    CONST robtarget p12664:= [[1532.1310620615823, -51.755404230859114, 1003.500033578516], [0, 0, 1, 0], [0, 0, 0, 0], [9E9, 9E9, 9E9, 9E9, 9E9, 9E9]];
    CONST robtarget p12665:= [[1531.2618371973992, -52.270415118434464, 1003.500033578516], [0, 0, 1, 0], [0, 0, 0, 0], [9E9, 9E9, 9E9, 9E9, 9E9, 9E9]];
    CONST robtarget p12666:= [[1530.6100576659546, -52.63207456238566, 1003.500033578516], [0, 0, 1, 0], [0, 0, 0, 0], [9E9, 9E9, 9E9, 9E9, 9E9, 9E9]];
    CONST robtarget p12667:= [[1530.2931638971058, -52.82618686460231, 1003.500033578516], [0, 0, 1, 0], [0, 0, 0, 0], [9E9, 9E9, 9E9, 9E9, 9E9, 9E9]];
    CONST robtarget p12668:= [[1529.7863810110655, -53.08892651938235, 1003.500033578516], [0, 0, 1, 0], [0, 0, 0, 0], [9E9, 9E9, 9E9, 9E9, 9E9, 9E9]];
    CONST robtarget p12669:= [[1529.7367415978995, -53.11810760441107, 1003.500033578516], [0, 0, 1, 0], [0, 0, 0, 0], [9E9, 9E9, 9E9, 9E9, 9E9, 9E9]];
    CONST robtarget p12670:= [[1529.1847719882317, -53.41718675288824, 1003.500033578516], [0, 0, 1, 0], [0, 0, 0, 0], [9E9, 9E9, 9E9, 9E9, 9E9, 9E9]];
    CONST robtarget p12671:= [[1528.9656328563278, -53.54211952816121, 1003.500033578516], [0, 0, 1, 0], [0, 0, 0, 0], [9E9, 9E9, 9E9, 9E9, 9E9, 9E9]];
    CONST robtarget p12672:= [[1528.4780900744865, -53.83944066606885, 1003.500033578516], [0, 0, 1, 0], [0, 0, 0, 0], [9E9, 9E9, 9E9, 9E9, 9E9, 9E9]];
    CONST robtarget p12673:= [[1527.6960366206135, -54.26689992615866, 1003.500033578516], [0, 0, 1, 0], [0, 0, 0, 0], [9E9, 9E9, 9E9, 9E9, 9E9, 9E9]];
    CONST robtarget p12674:= [[1527.2898060617083, -54.45592588754269, 1003.500033578516], [0, 0, 1, 0], [0, 0, 0, 0], [9E9, 9E9, 9E9, 9E9, 9E9, 9E9]];
    CONST robtarget p12675:= [[1526.7303787533363, -54.710685409871346, 1003.500033578516], [0, 0, 1, 0], [0, 0, 0, 0], [9E9, 9E9, 9E9, 9E9, 9E9, 9E9]];
    CONST robtarget p12676:= [[1526.1686464097916, -54.92872139464171, 1003.500033578516], [0, 0, 1, 0], [0, 0, 0, 0], [9E9, 9E9, 9E9, 9E9, 9E9, 9E9]];
    CONST robtarget p12677:= [[1525.7512622465076, -55.13249219015158, 1003.500033578516], [0, 0, 1, 0], [0, 0, 0, 0], [9E9, 9E9, 9E9, 9E9, 9E9, 9E9]];
    CONST robtarget p12678:= [[1525.1590179163616, -55.431827644455886, 1003.500033578516], [0, 0, 1, 0], [0, 0, 0, 0], [9E9, 9E9, 9E9, 9E9, 9E9, 9E9]];
    CONST robtarget p12679:= [[1525.0064466097315, -55.5144084202345, 1003.500033578516], [0, 0, 1, 0], [0, 0, 0, 0], [9E9, 9E9, 9E9, 9E9, 9E9, 9E9]];
    CONST robtarget p12680:= [[1524.838681406511, -55.59887141094046, 1003.500033578516], [0, 0, 1, 0], [0, 0, 0, 0], [9E9, 9E9, 9E9, 9E9, 9E9, 9E9]];
    CONST robtarget p12681:= [[1524.412701120568, -55.80300474395773, 1003.500033578516], [0, 0, 1, 0], [0, 0, 0, 0], [9E9, 9E9, 9E9, 9E9, 9E9, 9E9]];
    CONST robtarget p12682:= [[1523.8137863507948, -56.0413945246957, 1003.500033578516], [0, 0, 1, 0], [0, 0, 0, 0], [9E9, 9E9, 9E9, 9E9, 9E9, 9E9]];
    CONST robtarget p12683:= [[1523.096794661028, -56.341017791955295, 1003.500033578516], [0, 0, 1, 0], [0, 0, 0, 0], [9E9, 9E9, 9E9, 9E9, 9E9, 9E9]];
    CONST robtarget p12684:= [[1522.900783238865, -56.42082180491421, 1003.500033578516], [0, 0, 1, 0], [0, 0, 0, 0], [9E9, 9E9, 9E9, 9E9, 9E9, 9E9]];
    CONST robtarget p12685:= [[1522.6082814196384, -56.545971688333516, 1003.500033578516], [0, 0, 1, 0], [0, 0, 0, 0], [9E9, 9E9, 9E9, 9E9, 9E9, 9E9]];
    CONST robtarget p12686:= [[1522.1889282350046, -56.6709628567649, 1003.500033578516], [0, 0, 1, 0], [0, 0, 0, 0], [9E9, 9E9, 9E9, 9E9, 9E9, 9E9]];
    CONST robtarget p12687:= [[1521.3015503338331, -57.03764612699189, 1003.500033578516], [0, 0, 1, 0], [0, 0, 0, 0], [9E9, 9E9, 9E9, 9E9, 9E9, 9E9]];
    CONST robtarget p12688:= [[1520.80306051841, -57.23276139857534, 1003.500033578516], [0, 0, 1, 0], [0, 0, 0, 0], [9E9, 9E9, 9E9, 9E9, 9E9, 9E9]];
    CONST robtarget p12689:= [[1520.6617507120266, -57.27868779379712, 1003.500033578516], [0, 0, 1, 0], [0, 0, 0, 0], [9E9, 9E9, 9E9, 9E9, 9E9, 9E9]];
    CONST robtarget p12690:= [[1519.8184170172012, -57.589773311048475, 1003.500033578516], [0, 0, 1, 0], [0, 0, 0, 0], [9E9, 9E9, 9E9, 9E9, 9E9, 9E9]];
    CONST robtarget p12691:= [[1519.6469440456822, -57.65315375966382, 1003.500033578516], [0, 0, 1, 0], [0, 0, 0, 0], [9E9, 9E9, 9E9, 9E9, 9E9, 9E9]];
    CONST robtarget p12692:= [[1518.9672123317812, -57.88370126778568, 1003.500033578516], [0, 0, 1, 0], [0, 0, 0, 0], [9E9, 9E9, 9E9, 9E9, 9E9, 9E9]];
    CONST robtarget p12693:= [[1517.866507887685, -58.20960162710837, 1003.500033578516], [0, 0, 1, 0], [0, 0, 0, 0], [9E9, 9E9, 9E9, 9E9, 9E9, 9E9]];
    CONST robtarget p12694:= [[1517.564370643482, -58.28325027030423, 1003.500033578516], [0, 0, 1, 0], [0, 0, 0, 0], [9E9, 9E9, 9E9, 9E9, 9E9, 9E9]];
    CONST robtarget p12695:= [[1517.3151101543563, -58.359110977004875, 1003.500033578516], [0, 0, 1, 0], [0, 0, 0, 0], [9E9, 9E9, 9E9, 9E9, 9E9, 9E9]];
    CONST robtarget p12696:= [[1516.4046109578076, -58.64286422475155, 1003.500033578516], [0, 0, 1, 0], [0, 0, 0, 0], [9E9, 9E9, 9E9, 9E9, 9E9, 9E9]];
    CONST robtarget p12697:= [[1515.9569505437983, -58.768392762982955, 1003.500033578516], [0, 0, 1, 0], [0, 0, 0, 0], [9E9, 9E9, 9E9, 9E9, 9E9, 9E9]];
    CONST robtarget p12698:= [[1515.5151199352963, -58.91022808552202, 1003.500033578516], [0, 0, 1, 0], [0, 0, 0, 0], [9E9, 9E9, 9E9, 9E9, 9E9, 9E9]];
    CONST robtarget p12699:= [[1515.192527778176, -58.960963909001194, 1003.500033578516], [0, 0, 1, 0], [0, 0, 0, 0], [9E9, 9E9, 9E9, 9E9, 9E9, 9E9]];
    CONST robtarget p12700:= [[1514.1503402686096, -59.22694543179028, 1003.500033578516], [0, 0, 1, 0], [0, 0, 0, 0], [9E9, 9E9, 9E9, 9E9, 9E9, 9E9]];
    CONST robtarget p12701:= [[1513.5557447633169, -59.360352740508816, 1003.500033578516], [0, 0, 1, 0], [0, 0, 0, 0], [9E9, 9E9, 9E9, 9E9, 9E9, 9E9]];
    CONST robtarget p12702:= [[1513.2934993638064, -59.398941220659864, 1003.500033578516], [0, 0, 1, 0], [0, 0, 0, 0], [9E9, 9E9, 9E9, 9E9, 9E9, 9E9]];
    CONST robtarget p12703:= [[1512.403489281292, -59.608763300548, 1003.500033578516], [0, 0, 1, 0], [0, 0, 0, 0], [9E9, 9E9, 9E9, 9E9, 9E9, 9E9]];
    CONST robtarget p12704:= [[1512.0296429570128, -59.685111800334646, 1003.500033578516], [0, 0, 1, 0], [0, 0, 0, 0], [9E9, 9E9, 9E9, 9E9, 9E9, 9E9]];
    CONST robtarget p12705:= [[1511.4338776805575, -59.82476628793355, 1003.500033578516], [0, 0, 1, 0], [0, 0, 0, 0], [9E9, 9E9, 9E9, 9E9, 9E9, 9E9]];
    CONST robtarget p12706:= [[1510.9881098887731, -59.91814747321601, 1003.500033578516], [0, 0, 1, 0], [0, 0, 0, 0], [9E9, 9E9, 9E9, 9E9, 9E9, 9E9]];
    CONST robtarget p12707:= [[1510.8070079036906, -59.94973532784152, 1003.500033578516], [0, 0, 1, 0], [0, 0, 0, 0], [9E9, 9E9, 9E9, 9E9, 9E9, 9E9]];
    CONST robtarget p12708:= [[1510.7448277760268, -59.96038495608518, 1003.500033578516], [0, 0, 1, 0], [0, 0, 0, 0], [9E9, 9E9, 9E9, 9E9, 9E9, 9E9]];
    CONST robtarget p12709:= [[1510.4745015685621, -59.98646378804859, 1003.500033578516], [0, 0, 1, 0], [0, 0, 0, 0], [9E9, 9E9, 9E9, 9E9, 9E9, 9E9]];
    CONST robtarget p12710:= [[1510.0909268709627, -60.04140453241323, 1003.500033578516], [0, 0, 1, 0], [0, 0, 0, 0], [9E9, 9E9, 9E9, 9E9, 9E9, 9E9]];
    CONST robtarget p12711:= [[1509.4092115213996, -60.151023493626894, 1003.500033578516], [0, 0, 1, 0], [0, 0, 0, 0], [9E9, 9E9, 9E9, 9E9, 9E9, 9E9]];
    CONST robtarget p12712:= [[1509.1407802614508, -60.19882687326773, 1003.500033578516], [0, 0, 1, 0], [0, 0, 0, 0], [9E9, 9E9, 9E9, 9E9, 9E9, 9E9]];
    CONST robtarget p12713:= [[1508.5601837016875, -60.26340042336168, 1003.500033578516], [0, 0, 1, 0], [0, 0, 0, 0], [9E9, 9E9, 9E9, 9E9, 9E9, 9E9]];
    CONST robtarget p12714:= [[1507.6640295886964, -60.397835897292495, 1003.500033578516], [0, 0, 1, 0], [0, 0, 0, 0], [9E9, 9E9, 9E9, 9E9, 9E9, 9E9]];
    CONST robtarget p12715:= [[1507.3205366995528, -60.44744484086121, 1003.500033578516], [0, 0, 1, 0], [0, 0, 0, 0], [9E9, 9E9, 9E9, 9E9, 9E9, 9E9]];
    CONST robtarget p12716:= [[1506.9198397004645, -60.48554848075174, 1003.500033578516], [0, 0, 1, 0], [0, 0, 0, 0], [9E9, 9E9, 9E9, 9E9, 9E9, 9E9]];
    CONST robtarget p12717:= [[1506.3480021439116, -60.54932865497324, 1003.500033578516], [0, 0, 1, 0], [0, 0, 0, 0], [9E9, 9E9, 9E9, 9E9, 9E9, 9E9]];
    CONST robtarget p12718:= [[1506.0286245296538, -60.606260280640186, 1003.500033578516], [0, 0, 1, 0], [0, 0, 0, 0], [9E9, 9E9, 9E9, 9E9, 9E9, 9E9]];
    CONST robtarget p12719:= [[1505.9492369877419, -60.60951490106271, 1003.500033578516], [0, 0, 1, 0], [0, 0, 0, 0], [9E9, 9E9, 9E9, 9E9, 9E9, 9E9]];
    CONST robtarget p12720:= [[1505.8789526524727, -60.611009085656356, 1003.500033578516], [0, 0, 1, 0], [0, 0, 0, 0], [9E9, 9E9, 9E9, 9E9, 9E9, 9E9]];
    CONST robtarget p12721:= [[1505.3224203883021, -60.65045746650896, 1003.500033578516], [0, 0, 1, 0], [0, 0, 0, 0], [9E9, 9E9, 9E9, 9E9, 9E9, 9E9]];
    CONST robtarget p12722:= [[1505.1441541680317, -60.672558378263645, 1003.500033578516], [0, 0, 1, 0], [0, 0, 0, 0], [9E9, 9E9, 9E9, 9E9, 9E9, 9E9]];
    CONST robtarget p12723:= [[1504.3770680072512, -60.70421225380319, 1003.500033578516], [0, 0, 1, 0], [0, 0, 0, 0], [9E9, 9E9, 9E9, 9E9, 9E9, 9E9]];
    CONST robtarget p12724:= [[1503.8992364217452, -60.77229114782248, 1003.500033578516], [0, 0, 1, 0], [0, 0, 0, 0], [9E9, 9E9, 9E9, 9E9, 9E9, 9E9]];
    CONST robtarget p12725:= [[1503.093503312446, -60.829713664428, 1003.500033578516], [0, 0, 1, 0], [0, 0, 0, 0], [9E9, 9E9, 9E9, 9E9, 9E9, 9E9]];
    CONST robtarget p12726:= [[1502.275028322799, -60.865266701102776, 1003.500033578516], [0, 0, 1, 0], [0, 0, 0, 0], [9E9, 9E9, 9E9, 9E9, 9E9, 9E9]];
    CONST robtarget p12727:= [[1501.7502801780977, -60.87680720154429, 1003.500033578516], [0, 0, 1, 0], [0, 0, 0, 0], [9E9, 9E9, 9E9, 9E9, 9E9, 9E9]];
    CONST robtarget p12728:= [[1501.1321717850142, -60.86812155272374, 1003.500033578516], [0, 0, 1, 0], [0, 0, 0, 0], [9E9, 9E9, 9E9, 9E9, 9E9, 9E9]];
    CONST robtarget p12729:= [[1500.3650176022602, -60.89439954561838, 1003.500033578516], [0, 0, 1, 0], [0, 0, 0, 0], [9E9, 9E9, 9E9, 9E9, 9E9, 9E9]];
    CONST robtarget p12730:= [[1500.0005887741925, -60.88714554662218, 1003.500033578516], [0, 0, 1, 0], [0, 0, 0, 0], [9E9, 9E9, 9E9, 9E9, 9E9, 9E9]];
    CONST robtarget p12731:= [[1499.6330786731016, -60.86918679644523, 1003.500033578516], [0, 0, 1, 0], [0, 0, 0, 0], [9E9, 9E9, 9E9, 9E9, 9E9, 9E9]];
    CONST robtarget p12732:= [[1498.7343183829123, -60.89301213573544, 1003.500033578516], [0, 0, 1, 0], [0, 0, 0, 0], [9E9, 9E9, 9E9, 9E9, 9E9, 9E9]];
    CONST robtarget p12733:= [[1497.8384561952996, -60.879011023600654, 1003.500033578516], [0, 0, 1, 0], [0, 0, 0, 0], [9E9, 9E9, 9E9, 9E9, 9E9, 9E9]];
    CONST robtarget p12734:= [[1497.0922041448482, -60.83771003512446, 1003.500033578516], [0, 0, 1, 0], [0, 0, 0, 0], [9E9, 9E9, 9E9, 9E9, 9E9, 9E9]];
    CONST robtarget p12735:= [[1496.8361997453076, -60.82603686445868, 1003.500033578516], [0, 0, 1, 0], [0, 0, 0, 0], [9E9, 9E9, 9E9, 9E9, 9E9, 9E9]];
    CONST robtarget p12736:= [[1496.4138965917214, -60.778275502153924, 1003.500033578516], [0, 0, 1, 0], [0, 0, 0, 0], [9E9, 9E9, 9E9, 9E9, 9E9, 9E9]];
    CONST robtarget p12737:= [[1495.8035146590512, -60.74767869639028, 1003.500033578516], [0, 0, 1, 0], [0, 0, 0, 0], [9E9, 9E9, 9E9, 9E9, 9E9, 9E9]];
    CONST robtarget p12738:= [[1495.6187393990072, -60.72769177277266, 1003.500033578516], [0, 0, 1, 0], [0, 0, 0, 0], [9E9, 9E9, 9E9, 9E9, 9E9, 9E9]];
    CONST robtarget p12739:= [[1495.126932201303, -60.70252857016523, 1003.500033578516], [0, 0, 1, 0], [0, 0, 0, 0], [9E9, 9E9, 9E9, 9E9, 9E9, 9E9]];
    CONST robtarget p12740:= [[1494.505248273516, -60.640040835068014, 1003.500033578516], [0, 0, 1, 0], [0, 0, 0, 0], [9E9, 9E9, 9E9, 9E9, 9E9, 9E9]];
    CONST robtarget p12741:= [[1493.9707970922311, -60.586603258026315, 1003.500033578516], [0, 0, 1, 0], [0, 0, 0, 0], [9E9, 9E9, 9E9, 9E9, 9E9, 9E9]];
    CONST robtarget p12742:= [[1493.728122281413, -60.57869577579727, 1003.500033578516], [0, 0, 1, 0], [0, 0, 0, 0], [9E9, 9E9, 9E9, 9E9, 9E9, 9E9]];
    CONST robtarget p12743:= [[1493.3207496594594, -60.545796007754376, 1003.500033578516], [0, 0, 1, 0], [0, 0, 0, 0], [9E9, 9E9, 9E9, 9E9, 9E9, 9E9]];
    CONST robtarget p12744:= [[1493.0342588648045, -60.515907015423046, 1003.500033578516], [0, 0, 1, 0], [0, 0, 0, 0], [9E9, 9E9, 9E9, 9E9, 9E9, 9E9]];
    CONST robtarget p12745:= [[1492.5314490561839, -60.42360355630814, 1003.500033578516], [0, 0, 1, 0], [0, 0, 0, 0], [9E9, 9E9, 9E9, 9E9, 9E9, 9E9]];
    CONST robtarget p12746:= [[1491.6668361516013, -60.32164521258506, 1003.500033578516], [0, 0, 1, 0], [0, 0, 0, 0], [9E9, 9E9, 9E9, 9E9, 9E9, 9E9]];
    CONST robtarget p12747:= [[1490.7479630489497, -60.18407184896695, 1003.500033578516], [0, 0, 1, 0], [0, 0, 0, 0], [9E9, 9E9, 9E9, 9E9, 9E9, 9E9]];
    CONST robtarget p12748:= [[1489.9914983282804, -60.0648048675663, 1003.500033578516], [0, 0, 1, 0], [0, 0, 0, 0], [9E9, 9E9, 9E9, 9E9, 9E9, 9E9]];
    CONST robtarget p12749:= [[1489.8132747932655, -60.050032149975266, 1003.500033578516], [0, 0, 1, 0], [0, 0, 0, 0], [9E9, 9E9, 9E9, 9E9, 9E9, 9E9]];
    CONST robtarget p12750:= [[1489.6954944579838, -60.02336426978388, 1003.500033578516], [0, 0, 1, 0], [0, 0, 0, 0], [9E9, 9E9, 9E9, 9E9, 9E9, 9E9]];
    CONST robtarget p12751:= [[1489.2307032090532, -59.94463917957851, 1003.500033578516], [0, 0, 1, 0], [0, 0, 0, 0], [9E9, 9E9, 9E9, 9E9, 9E9, 9E9]];
    CONST robtarget p12752:= [[1488.969375621922, -59.912737352572954, 1003.500033578516], [0, 0, 1, 0], [0, 0, 0, 0], [9E9, 9E9, 9E9, 9E9, 9E9, 9E9]];
    CONST robtarget p12753:= [[1488.212151107269, -59.73070325446558, 1003.500033578516], [0, 0, 1, 0], [0, 0, 0, 0], [9E9, 9E9, 9E9, 9E9, 9E9, 9E9]];
    CONST robtarget p12754:= [[1487.9882544856496, -59.699601630604995, 1003.500033578516], [0, 0, 1, 0], [0, 0, 0, 0], [9E9, 9E9, 9E9, 9E9, 9E9, 9E9]];
    CONST robtarget p12755:= [[1487.9148646222939, -59.6846132005301, 1003.500033578516], [0, 0, 1, 0], [0, 0, 0, 0], [9E9, 9E9, 9E9, 9E9, 9E9, 9E9]];
    CONST robtarget p12756:= [[1486.6279582909926, -59.37969541445614, 1003.500033578516], [0, 0, 1, 0], [0, 0, 0, 0], [9E9, 9E9, 9E9, 9E9, 9E9, 9E9]];
    CONST robtarget p12757:= [[1486.140888283754, -59.292200601364186, 1003.500033578516], [0, 0, 1, 0], [0, 0, 0, 0], [9E9, 9E9, 9E9, 9E9, 9E9, 9E9]];
    CONST robtarget p12758:= [[1485.6944591473587, -59.19830148713572, 1003.500033578516], [0, 0, 1, 0], [0, 0, 0, 0], [9E9, 9E9, 9E9, 9E9, 9E9, 9E9]];
    CONST robtarget p12759:= [[1484.794375410712, -58.99350436981834, 1003.500033578516], [0, 0, 1, 0], [0, 0, 0, 0], [9E9, 9E9, 9E9, 9E9, 9E9, 9E9]];
    CONST robtarget p12760:= [[1484.3195121421352, -58.82802177044728, 1003.500033578516], [0, 0, 1, 0], [0, 0, 0, 0], [9E9, 9E9, 9E9, 9E9, 9E9, 9E9]];
    CONST robtarget p12761:= [[1483.608527363885, -58.63685731582685, 1003.500033578516], [0, 0, 1, 0], [0, 0, 0, 0], [9E9, 9E9, 9E9, 9E9, 9E9, 9E9]];
    CONST robtarget p12762:= [[1483.46717818544, -58.58551762263184, 1003.500033578516], [0, 0, 1, 0], [0, 0, 0, 0], [9E9, 9E9, 9E9, 9E9, 9E9, 9E9]];
    CONST robtarget p12763:= [[1482.7397918590495, -58.37344401868633, 1003.500033578516], [0, 0, 1, 0], [0, 0, 0, 0], [9E9, 9E9, 9E9, 9E9, 9E9, 9E9]];
    CONST robtarget p12764:= [[1482.3591697778888, -58.2723436864768, 1003.500033578516], [0, 0, 1, 0], [0, 0, 0, 0], [9E9, 9E9, 9E9, 9E9, 9E9, 9E9]];
    CONST robtarget p12765:= [[1481.8585054728746, -58.11198192141396, 1003.500033578516], [0, 0, 1, 0], [0, 0, 0, 0], [9E9, 9E9, 9E9, 9E9, 9E9, 9E9]];
    CONST robtarget p12766:= [[1481.3685817283563, -57.93737088101702, 1003.500033578516], [0, 0, 1, 0], [0, 0, 0, 0], [9E9, 9E9, 9E9, 9E9, 9E9, 9E9]];
    CONST robtarget p12767:= [[1480.6995920486086, -57.765830924699586, 1003.500033578516], [0, 0, 1, 0], [0, 0, 0, 0], [9E9, 9E9, 9E9, 9E9, 9E9, 9E9]];
    CONST robtarget p12768:= [[1480.3436933161818, -57.66286123975082, 1003.500033578516], [0, 0, 1, 0], [0, 0, 0, 0], [9E9, 9E9, 9E9, 9E9, 9E9, 9E9]];
    CONST robtarget p12769:= [[1479.9731860993122, -57.540607606285775, 1003.500033578516], [0, 0, 1, 0], [0, 0, 0, 0], [9E9, 9E9, 9E9, 9E9, 9E9, 9E9]];
    CONST robtarget p12770:= [[1479.7781265101073, -57.45151979305535, 1003.500033578516], [0, 0, 1, 0], [0, 0, 0, 0], [9E9, 9E9, 9E9, 9E9, 9E9, 9E9]];
    CONST robtarget p12771:= [[1479.4149893289998, -57.307912593364954, 1003.500033578516], [0, 0, 1, 0], [0, 0, 0, 0], [9E9, 9E9, 9E9, 9E9, 9E9, 9E9]];
    CONST robtarget p12772:= [[1479.218654376944, -57.23642583891754, 1003.500033578516], [0, 0, 1, 0], [0, 0, 0, 0], [9E9, 9E9, 9E9, 9E9, 9E9, 9E9]];
    CONST robtarget p12773:= [[1478.7985262864372, -57.06718631801597, 1003.500033578516], [0, 0, 1, 0], [0, 0, 0, 0], [9E9, 9E9, 9E9, 9E9, 9E9, 9E9]];
    CONST robtarget p12774:= [[1478.4967717020684, -56.966101153962924, 1003.500033578516], [0, 0, 1, 0], [0, 0, 0, 0], [9E9, 9E9, 9E9, 9E9, 9E9, 9E9]];
    CONST robtarget p12775:= [[1478.0783051864335, -56.80894886473797, 1003.500033578516], [0, 0, 1, 0], [0, 0, 0, 0], [9E9, 9E9, 9E9, 9E9, 9E9, 9E9]];
    CONST robtarget p12776:= [[1477.8972557411332, -56.73871748054797, 1003.500033578516], [0, 0, 1, 0], [0, 0, 0, 0], [9E9, 9E9, 9E9, 9E9, 9E9, 9E9]];
    CONST robtarget p12777:= [[1477.419040496479, -56.55728204433218, 1003.500033578516], [0, 0, 1, 0], [0, 0, 0, 0], [9E9, 9E9, 9E9, 9E9, 9E9, 9E9]];
    CONST robtarget p12778:= [[1477.0224585378432, -56.40800549919932, 1003.500033578516], [0, 0, 1, 0], [0, 0, 0, 0], [9E9, 9E9, 9E9, 9E9, 9E9, 9E9]];
    CONST robtarget p12779:= [[1476.6457873835752, -56.25716671121214, 1003.500033578516], [0, 0, 1, 0], [0, 0, 0, 0], [9E9, 9E9, 9E9, 9E9, 9E9, 9E9]];
    CONST robtarget p12780:= [[1476.3107290898254, -56.11531359924879, 1003.500033578516], [0, 0, 1, 0], [0, 0, 0, 0], [9E9, 9E9, 9E9, 9E9, 9E9, 9E9]];
    CONST robtarget p12781:= [[1475.757101201903, -55.857580148854815, 1003.500033578516], [0, 0, 1, 0], [0, 0, 0, 0], [9E9, 9E9, 9E9, 9E9, 9E9, 9E9]];
    CONST robtarget p12782:= [[1475.2412390471118, -55.63567586356051, 1003.500033578516], [0, 0, 1, 0], [0, 0, 0, 0], [9E9, 9E9, 9E9, 9E9, 9E9, 9E9]];
    CONST robtarget p12783:= [[1474.739043483524, -55.405277609739095, 1003.500033578516], [0, 0, 1, 0], [0, 0, 0, 0], [9E9, 9E9, 9E9, 9E9, 9E9, 9E9]];
    CONST robtarget p12784:= [[1474.0668552668544, -55.09690623872325, 1003.500033578516], [0, 0, 1, 0], [0, 0, 0, 0], [9E9, 9E9, 9E9, 9E9, 9E9, 9E9]];
    CONST robtarget p12785:= [[1473.385601323675, -54.7780424045763, 1003.500033578516], [0, 0, 1, 0], [0, 0, 0, 0], [9E9, 9E9, 9E9, 9E9, 9E9, 9E9]];
    CONST robtarget p12786:= [[1472.9079373070804, -54.55434300745352, 1003.500033578516], [0, 0, 1, 0], [0, 0, 0, 0], [9E9, 9E9, 9E9, 9E9, 9E9, 9E9]];
    CONST robtarget p12787:= [[1472.6979268486778, -54.442761967229664, 1003.500033578516], [0, 0, 1, 0], [0, 0, 0, 0], [9E9, 9E9, 9E9, 9E9, 9E9, 9E9]];
    CONST robtarget p12788:= [[1472.5192556122183, -54.356856623518055, 1003.500033578516], [0, 0, 1, 0], [0, 0, 0, 0], [9E9, 9E9, 9E9, 9E9, 9E9, 9E9]];
    CONST robtarget p12789:= [[1472.3433857548564, -54.276293800346956, 1003.500033578516], [0, 0, 1, 0], [0, 0, 0, 0], [9E9, 9E9, 9E9, 9E9, 9E9, 9E9]];
    CONST robtarget p12790:= [[1471.6735811086735, -53.90700087718467, 1003.500033578516], [0, 0, 1, 0], [0, 0, 0, 0], [9E9, 9E9, 9E9, 9E9, 9E9, 9E9]];
    CONST robtarget p12791:= [[1471.6118633825038, -53.878311391837045, 1003.500033578516], [0, 0, 1, 0], [0, 0, 0, 0], [9E9, 9E9, 9E9, 9E9, 9E9, 9E9]];
    CONST robtarget p12792:= [[1470.9147178970193, -53.45979797031765, 1003.500033578516], [0, 0, 1, 0], [0, 0, 0, 0], [9E9, 9E9, 9E9, 9E9, 9E9, 9E9]];
    CONST robtarget p12793:= [[1470.3308377490243, -53.15743980218656, 1003.500033578516], [0, 0, 1, 0], [0, 0, 0, 0], [9E9, 9E9, 9E9, 9E9, 9E9, 9E9]];
    CONST robtarget p12794:= [[1469.981792326095, -52.947352811709806, 1003.500033578516], [0, 0, 1, 0], [0, 0, 0, 0], [9E9, 9E9, 9E9, 9E9, 9E9, 9E9]];
    CONST robtarget p12795:= [[1469.739501525089, -52.80895313601386, 1003.500033578516], [0, 0, 1, 0], [0, 0, 0, 0], [9E9, 9E9, 9E9, 9E9, 9E9, 9E9]];
    CONST robtarget p12796:= [[1469.041702666435, -52.44123634005517, 1003.500033578516], [0, 0, 1, 0], [0, 0, 0, 0], [9E9, 9E9, 9E9, 9E9, 9E9, 9E9]];
    CONST robtarget p12797:= [[1468.8959017630361, -52.36046703095187, 1003.500033578516], [0, 0, 1, 0], [0, 0, 0, 0], [9E9, 9E9, 9E9, 9E9, 9E9, 9E9]];
    CONST robtarget p12798:= [[1468.4325252838353, -52.0869439815557, 1003.500033578516], [0, 0, 1, 0], [0, 0, 0, 0], [9E9, 9E9, 9E9, 9E9, 9E9, 9E9]];
    CONST robtarget p12799:= [[1468.1673742737253, -51.94219004913117, 1003.500033578516], [0, 0, 1, 0], [0, 0, 0, 0], [9E9, 9E9, 9E9, 9E9, 9E9, 9E9]];
    CONST robtarget p12800:= [[1467.8230360238244, -51.71098401292481, 1003.500033578516], [0, 0, 1, 0], [0, 0, 0, 0], [9E9, 9E9, 9E9, 9E9, 9E9, 9E9]];
    CONST robtarget p12801:= [[1467.2709033189144, -51.358364491315115, 1003.500033578516], [0, 0, 1, 0], [0, 0, 0, 0], [9E9, 9E9, 9E9, 9E9, 9E9, 9E9]];
    CONST robtarget p12802:= [[1466.8163805918425, -51.06205975062079, 1003.500033578516], [0, 0, 1, 0], [0, 0, 0, 0], [9E9, 9E9, 9E9, 9E9, 9E9, 9E9]];
    CONST robtarget p12803:= [[1466.3285514799147, -50.71988024332508, 1003.500033578516], [0, 0, 1, 0], [0, 0, 0, 0], [9E9, 9E9, 9E9, 9E9, 9E9, 9E9]];
    CONST robtarget p12804:= [[1466.0550435531595, -50.560233816038036, 1003.500033578516], [0, 0, 1, 0], [0, 0, 0, 0], [9E9, 9E9, 9E9, 9E9, 9E9, 9E9]];
    CONST robtarget p12805:= [[1465.7588315671217, -50.344417835721075, 1003.500033578516], [0, 0, 1, 0], [0, 0, 0, 0], [9E9, 9E9, 9E9, 9E9, 9E9, 9E9]];
    CONST robtarget p12806:= [[1465.2675983109084, -50.03925991860115, 1003.500033578516], [0, 0, 1, 0], [0, 0, 0, 0], [9E9, 9E9, 9E9, 9E9, 9E9, 9E9]];
    CONST robtarget p12807:= [[1464.3223192555545, -49.37751525942017, 1003.500033578516], [0, 0, 1, 0], [0, 0, 0, 0], [9E9, 9E9, 9E9, 9E9, 9E9, 9E9]];
    CONST robtarget p12808:= [[1464.12423373144, -49.238278317764404, 1003.500033578516], [0, 0, 1, 0], [0, 0, 0, 0], [9E9, 9E9, 9E9, 9E9, 9E9, 9E9]];
    CONST robtarget p12809:= [[1463.7933652636184, -48.94931296831757, 1003.500033578516], [0, 0, 1, 0], [0, 0, 0, 0], [9E9, 9E9, 9E9, 9E9, 9E9, 9E9]];
    CONST robtarget p12810:= [[1463.7214730998505, -48.887040437062296, 1003.500033578516], [0, 0, 1, 0], [0, 0, 0, 0], [9E9, 9E9, 9E9, 9E9, 9E9, 9E9]];
    CONST robtarget p12811:= [[1463.5352670470895, -48.735788801459876, 1003.500033578516], [0, 0, 1, 0], [0, 0, 0, 0], [9E9, 9E9, 9E9, 9E9, 9E9, 9E9]];
    CONST robtarget p12812:= [[1463.2784718498417, -48.53173457494182, 1003.500033578516], [0, 0, 1, 0], [0, 0, 0, 0], [9E9, 9E9, 9E9, 9E9, 9E9, 9E9]];
    CONST robtarget p12813:= [[1462.9332169287038, -48.26569111040662, 1003.500033578516], [0, 0, 1, 0], [0, 0, 0, 0], [9E9, 9E9, 9E9, 9E9, 9E9, 9E9]];
    CONST robtarget p12814:= [[1462.2842150312945, -47.816391831952515, 1003.500033578516], [0, 0, 1, 0], [0, 0, 0, 0], [9E9, 9E9, 9E9, 9E9, 9E9, 9E9]];
    CONST robtarget p12815:= [[1461.986972846843, -47.53643179228948, 1003.500033578516], [0, 0, 1, 0], [0, 0, 0, 0], [9E9, 9E9, 9E9, 9E9, 9E9, 9E9]];
    CONST robtarget p12816:= [[1461.7300433845637, -47.3279367766886, 1003.500033578516], [0, 0, 1, 0], [0, 0, 0, 0], [9E9, 9E9, 9E9, 9E9, 9E9, 9E9]];
    CONST robtarget p12817:= [[1461.3369768589682, -47.03757991187973, 1003.500033578516], [0, 0, 1, 0], [0, 0, 0, 0], [9E9, 9E9, 9E9, 9E9, 9E9, 9E9]];
    CONST robtarget p12818:= [[1461.136355692275, -46.893446375038046, 1003.500033578516], [0, 0, 1, 0], [0, 0, 0, 0], [9E9, 9E9, 9E9, 9E9, 9E9, 9E9]];
    CONST robtarget p12819:= [[1460.5447343118615, -46.40482173427037, 1003.500033578516], [0, 0, 1, 0], [0, 0, 0, 0], [9E9, 9E9, 9E9, 9E9, 9E9, 9E9]];
    CONST robtarget p12820:= [[1460.468501722416, -46.34424538688958, 1003.500033578516], [0, 0, 1, 0], [0, 0, 0, 0], [9E9, 9E9, 9E9, 9E9, 9E9, 9E9]];
    CONST robtarget p12821:= [[1460.0126248245635, -45.92682407313298, 1003.500033578516], [0, 0, 1, 0], [0, 0, 0, 0], [9E9, 9E9, 9E9, 9E9, 9E9, 9E9]];
    CONST robtarget p12822:= [[1459.8964465299503, -45.82845734358974, 1003.500033578516], [0, 0, 1, 0], [0, 0, 0, 0], [9E9, 9E9, 9E9, 9E9, 9E9, 9E9]];
    CONST robtarget p12823:= [[1459.4077100073077, -45.37554272869181, 1003.500033578516], [0, 0, 1, 0], [0, 0, 0, 0], [9E9, 9E9, 9E9, 9E9, 9E9, 9E9]];
    CONST robtarget p12824:= [[1459.1356373451918, -45.13210794821709, 1003.500033578516], [0, 0, 1, 0], [0, 0, 0, 0], [9E9, 9E9, 9E9, 9E9, 9E9, 9E9]];
    CONST robtarget p12825:= [[1458.833138050238, -44.83978029856981, 1003.500033578516], [0, 0, 1, 0], [0, 0, 0, 0], [9E9, 9E9, 9E9, 9E9, 9E9, 9E9]];
    CONST robtarget p12826:= [[1458.3208884897697, -44.383168360812384, 1003.500033578516], [0, 0, 1, 0], [0, 0, 0, 0], [9E9, 9E9, 9E9, 9E9, 9E9, 9E9]];
    CONST robtarget p12827:= [[1458.0020018869243, -44.10775357409478, 1003.500033578516], [0, 0, 1, 0], [0, 0, 0, 0], [9E9, 9E9, 9E9, 9E9, 9E9, 9E9]];
    CONST robtarget p12828:= [[1457.5682916572557, -43.71039476711136, 1003.500033578516], [0, 0, 1, 0], [0, 0, 0, 0], [9E9, 9E9, 9E9, 9E9, 9E9, 9E9]];
    CONST robtarget p12829:= [[1457.3426791650818, -43.47299808350768, 1003.500033578516], [0, 0, 1, 0], [0, 0, 0, 0], [9E9, 9E9, 9E9, 9E9, 9E9, 9E9]];
    CONST robtarget p12830:= [[1456.1648467534328, -42.27347390301688, 1003.500033578516], [0, 0, 1, 0], [0, 0, 0, 0], [9E9, 9E9, 9E9, 9E9, 9E9, 9E9]];
    CONST robtarget p12831:= [[1455.731171856514, -41.80753749343266, 1003.500033578516], [0, 0, 1, 0], [0, 0, 0, 0], [9E9, 9E9, 9E9, 9E9, 9E9, 9E9]];
    CONST robtarget p12832:= [[1455.4291936774002, -41.49946635981109, 1003.500033578516], [0, 0, 1, 0], [0, 0, 0, 0], [9E9, 9E9, 9E9, 9E9, 9E9, 9E9]];
    CONST robtarget p12833:= [[1455.1887223337912, -41.24203708161639, 1003.500033578516], [0, 0, 1, 0], [0, 0, 0, 0], [9E9, 9E9, 9E9, 9E9, 9E9, 9E9]];
    CONST robtarget p12834:= [[1454.657424573964, -40.677391201593565, 1003.500033578516], [0, 0, 1, 0], [0, 0, 0, 0], [9E9, 9E9, 9E9, 9E9, 9E9, 9E9]];
    CONST robtarget p12835:= [[1454.3013815324605, -40.24428470275707, 1003.500033578516], [0, 0, 1, 0], [0, 0, 0, 0], [9E9, 9E9, 9E9, 9E9, 9E9, 9E9]];
    CONST robtarget p12836:= [[1453.942913642316, -39.83943990642383, 1003.500033578516], [0, 0, 1, 0], [0, 0, 0, 0], [9E9, 9E9, 9E9, 9E9, 9E9, 9E9]];
    CONST robtarget p12837:= [[1453.5938907294917, -39.40632777756997, 1003.500033578516], [0, 0, 1, 0], [0, 0, 0, 0], [9E9, 9E9, 9E9, 9E9, 9E9, 9E9]];
    CONST robtarget p12838:= [[1453.477586969693, -39.28148252377899, 1003.500033578516], [0, 0, 1, 0], [0, 0, 0, 0], [9E9, 9E9, 9E9, 9E9, 9E9, 9E9]];
    CONST robtarget p12839:= [[1453.333997610336, -39.10047869658248, 1003.500033578516], [0, 0, 1, 0], [0, 0, 0, 0], [9E9, 9E9, 9E9, 9E9, 9E9, 9E9]];
    CONST robtarget p12840:= [[1453.0266983458246, -38.713415468882886, 1003.500033578516], [0, 0, 1, 0], [0, 0, 0, 0], [9E9, 9E9, 9E9, 9E9, 9E9, 9E9]];
    CONST robtarget p12841:= [[1452.5568761578324, -38.189069118549625, 1003.500033578516], [0, 0, 1, 0], [0, 0, 0, 0], [9E9, 9E9, 9E9, 9E9, 9E9, 9E9]];
    CONST robtarget p12842:= [[1452.3909681262012, -37.94822534388772, 1003.500033578516], [0, 0, 1, 0], [0, 0, 0, 0], [9E9, 9E9, 9E9, 9E9, 9E9, 9E9]];
    CONST robtarget p12843:= [[1452.0362579306045, -37.516652114643605, 1003.500033578516], [0, 0, 1, 0], [0, 0, 0, 0], [9E9, 9E9, 9E9, 9E9, 9E9, 9E9]];
    CONST robtarget p12844:= [[1451.9290080425333, -37.40084552126697, 1003.500033578516], [0, 0, 1, 0], [0, 0, 0, 0], [9E9, 9E9, 9E9, 9E9, 9E9, 9E9]];
    CONST robtarget p12845:= [[1451.6911292281357, -37.137695760035115, 1003.500033578516], [0, 0, 1, 0], [0, 0, 0, 0], [9E9, 9E9, 9E9, 9E9, 9E9, 9E9]];
    CONST robtarget p12846:= [[1451.5154365823112, -36.86592243989559, 1003.500033578516], [0, 0, 1, 0], [0, 0, 0, 0], [9E9, 9E9, 9E9, 9E9, 9E9, 9E9]];
    CONST robtarget p12847:= [[1451.1629200760685, -36.34540489414617, 1003.500033578516], [0, 0, 1, 0], [0, 0, 0, 0], [9E9, 9E9, 9E9, 9E9, 9E9, 9E9]];
    CONST robtarget p12848:= [[1450.8847145526963, -36.01049249746095, 1003.500033578516], [0, 0, 1, 0], [0, 0, 0, 0], [9E9, 9E9, 9E9, 9E9, 9E9, 9E9]];
    CONST robtarget p12849:= [[1450.6126521402598, -35.63256960029754, 1003.500033578516], [0, 0, 1, 0], [0, 0, 0, 0], [9E9, 9E9, 9E9, 9E9, 9E9, 9E9]];
    CONST robtarget p12850:= [[1450.4790397815684, -35.41322576066054, 1003.500033578516], [0, 0, 1, 0], [0, 0, 0, 0], [9E9, 9E9, 9E9, 9E9, 9E9, 9E9]];
    CONST robtarget p12851:= [[1450.0342587071136, -34.79318059085137, 1003.500033578516], [0, 0, 1, 0], [0, 0, 0, 0], [9E9, 9E9, 9E9, 9E9, 9E9, 9E9]];
    CONST robtarget p12852:= [[1449.8970297442795, -34.62186807893758, 1003.500033578516], [0, 0, 1, 0], [0, 0, 0, 0], [9E9, 9E9, 9E9, 9E9, 9E9, 9E9]];
    CONST robtarget p12853:= [[1449.4105252565382, -33.94793724110956, 1003.500033578516], [0, 0, 1, 0], [0, 0, 0, 0], [9E9, 9E9, 9E9, 9E9, 9E9, 9E9]];
    CONST robtarget p12854:= [[1449.1728074548507, -33.592148510738745, 1003.500033578516], [0, 0, 1, 0], [0, 0, 0, 0], [9E9, 9E9, 9E9, 9E9, 9E9, 9E9]];
    CONST robtarget p12855:= [[1448.7053989915553, -32.82032148636057, 1003.500033578516], [0, 0, 1, 0], [0, 0, 0, 0], [9E9, 9E9, 9E9, 9E9, 9E9, 9E9]];
    CONST robtarget p12856:= [[1448.6197802401284, -32.68049050813628, 1003.500033578516], [0, 0, 1, 0], [0, 0, 0, 0], [9E9, 9E9, 9E9, 9E9, 9E9, 9E9]];
    CONST robtarget p12857:= [[1448.3155348955765, -32.21672512372758, 1003.500033578516], [0, 0, 1, 0], [0, 0, 0, 0], [9E9, 9E9, 9E9, 9E9, 9E9, 9E9]];
    CONST robtarget p12858:= [[1447.8357512844905, -31.41441451551305, 1003.500033578516], [0, 0, 1, 0], [0, 0, 0, 0], [9E9, 9E9, 9E9, 9E9, 9E9, 9E9]];
    CONST robtarget p12859:= [[1447.6088591171, -31.024228994559174, 1003.500033578516], [0, 0, 1, 0], [0, 0, 0, 0], [9E9, 9E9, 9E9, 9E9, 9E9, 9E9]];
    CONST robtarget p12860:= [[1447.177998953813, -30.32372215622891, 1003.500033578516], [0, 0, 1, 0], [0, 0, 0, 0], [9E9, 9E9, 9E9, 9E9, 9E9, 9E9]];
    CONST robtarget p12861:= [[1447.08175185569, -30.140892856360814, 1003.500033578516], [0, 0, 1, 0], [0, 0, 0, 0], [9E9, 9E9, 9E9, 9E9, 9E9, 9E9]];
    CONST robtarget p12862:= [[1446.745962923399, -29.59670386966831, 1003.500033578516], [0, 0, 1, 0], [0, 0, 0, 0], [9E9, 9E9, 9E9, 9E9, 9E9, 9E9]];
    CONST robtarget p12863:= [[1446.5390177811498, -29.131187672454786, 1003.500033578516], [0, 0, 1, 0], [0, 0, 0, 0], [9E9, 9E9, 9E9, 9E9, 9E9, 9E9]];
    CONST robtarget p12864:= [[1446.4229958311491, -28.889432365324758, 1003.500033578516], [0, 0, 1, 0], [0, 0, 0, 0], [9E9, 9E9, 9E9, 9E9, 9E9, 9E9]];
    CONST robtarget p12865:= [[1446.176233251719, -28.455299744372766, 1003.500033578516], [0, 0, 1, 0], [0, 0, 0, 0], [9E9, 9E9, 9E9, 9E9, 9E9, 9E9]];
    CONST robtarget p12866:= [[1446.1164445218433, -28.33208788449391, 1003.500033578516], [0, 0, 1, 0], [0, 0, 0, 0], [9E9, 9E9, 9E9, 9E9, 9E9, 9E9]];
    CONST robtarget p12867:= [[1445.8132754479857, -27.77148556011396, 1003.500033578516], [0, 0, 1, 0], [0, 0, 0, 0], [9E9, 9E9, 9E9, 9E9, 9E9, 9E9]];
    CONST robtarget p12868:= [[1445.505302048922, -27.182220087026074, 1003.500033578516], [0, 0, 1, 0], [0, 0, 0, 0], [9E9, 9E9, 9E9, 9E9, 9E9, 9E9]];
    CONST robtarget p12869:= [[1445.3734843202117, -26.93806999737037, 1003.500033578516], [0, 0, 1, 0], [0, 0, 0, 0], [9E9, 9E9, 9E9, 9E9, 9E9, 9E9]];
    CONST robtarget p12870:= [[1445.2434851205492, -26.688133101147436, 1003.500033578516], [0, 0, 1, 0], [0, 0, 0, 0], [9E9, 9E9, 9E9, 9E9, 9E9, 9E9]];
    CONST robtarget p12871:= [[1444.9995996425355, -26.197629289649633, 1003.500033578516], [0, 0, 1, 0], [0, 0, 0, 0], [9E9, 9E9, 9E9, 9E9, 9E9, 9E9]];
    CONST robtarget p12872:= [[1444.817726879173, -25.788460106516965, 1003.500033578516], [0, 0, 1, 0], [0, 0, 0, 0], [9E9, 9E9, 9E9, 9E9, 9E9, 9E9]];
    CONST robtarget p12873:= [[1444.751989881604, -25.60082571060748, 1003.500033578516], [0, 0, 1, 0], [0, 0, 0, 0], [9E9, 9E9, 9E9, 9E9, 9E9, 9E9]];
    CONST robtarget p12874:= [[1444.4434203301457, -24.90798318354797, 1003.500033578516], [0, 0, 1, 0], [0, 0, 0, 0], [9E9, 9E9, 9E9, 9E9, 9E9, 9E9]];
    CONST robtarget p12875:= [[1444.250501272772, -24.4984780338729, 1003.500033578516], [0, 0, 1, 0], [0, 0, 0, 0], [9E9, 9E9, 9E9, 9E9, 9E9, 9E9]];
    CONST robtarget p12876:= [[1444.0499465487433, -24.013967825751152, 1003.500033578516], [0, 0, 1, 0], [0, 0, 0, 0], [9E9, 9E9, 9E9, 9E9, 9E9, 9E9]];
    CONST robtarget p12877:= [[1443.7685367007648, -23.375679640501296, 1003.500033578516], [0, 0, 1, 0], [0, 0, 0, 0], [9E9, 9E9, 9E9, 9E9, 9E9, 9E9]];
    CONST robtarget p12878:= [[1443.5016920450676, -22.761836486064702, 1003.500033578516], [0, 0, 1, 0], [0, 0, 0, 0], [9E9, 9E9, 9E9, 9E9, 9E9, 9E9]];
    CONST robtarget p12879:= [[1443.354463409008, -22.373718230581325, 1003.500033578516], [0, 0, 1, 0], [0, 0, 0, 0], [9E9, 9E9, 9E9, 9E9, 9E9, 9E9]];
    CONST robtarget p12880:= [[1443.0923587075204, -21.800190844486615, 1003.500033578516], [0, 0, 1, 0], [0, 0, 0, 0], [9E9, 9E9, 9E9, 9E9, 9E9, 9E9]];
    CONST robtarget p12881:= [[1442.9522374043968, -21.355280382477325, 1003.500033578516], [0, 0, 1, 0], [0, 0, 0, 0], [9E9, 9E9, 9E9, 9E9, 9E9, 9E9]];
    CONST robtarget p12882:= [[1442.7898385738413, -20.810125837381484, 1003.500033578516], [0, 0, 1, 0], [0, 0, 0, 0], [9E9, 9E9, 9E9, 9E9, 9E9, 9E9]];
    CONST robtarget p12883:= [[1442.6428254127886, -20.414595161209782, 1003.500033578516], [0, 0, 1, 0], [0, 0, 0, 0], [9E9, 9E9, 9E9, 9E9, 9E9, 9E9]];
    CONST robtarget p12884:= [[1442.3338227488105, -19.493724879034005, 1003.500033578516], [0, 0, 1, 0], [0, 0, 0, 0], [9E9, 9E9, 9E9, 9E9, 9E9, 9E9]];
    CONST robtarget p12885:= [[1442.215925822188, -19.172290044542756, 1003.500033578516], [0, 0, 1, 0], [0, 0, 0, 0], [9E9, 9E9, 9E9, 9E9, 9E9, 9E9]];
    CONST robtarget p12886:= [[1441.9701192981086, -18.512260769527572, 1003.500033578516], [0, 0, 1, 0], [0, 0, 0, 0], [9E9, 9E9, 9E9, 9E9, 9E9, 9E9]];
    CONST robtarget p12887:= [[1441.8283529618873, -17.9740752161238, 1003.500033578516], [0, 0, 1, 0], [0, 0, 0, 0], [9E9, 9E9, 9E9, 9E9, 9E9, 9E9]];
    CONST robtarget p12888:= [[1441.4771606448508, -16.925346029536627, 1003.500033578516], [0, 0, 1, 0], [0, 0, 0, 0], [9E9, 9E9, 9E9, 9E9, 9E9, 9E9]];
    CONST robtarget p12889:= [[1441.2720339694588, -16.028284145260898, 1003.500033578516], [0, 0, 1, 0], [0, 0, 0, 0], [9E9, 9E9, 9E9, 9E9, 9E9, 9E9]];
    CONST robtarget p12890:= [[1441.1449885887441, -15.639845525111049, 1003.500033578516], [0, 0, 1, 0], [0, 0, 0, 0], [9E9, 9E9, 9E9, 9E9, 9E9, 9E9]];
    CONST robtarget p12891:= [[1441.000430709358, -14.933612353946813, 1003.500033578516], [0, 0, 1, 0], [0, 0, 0, 0], [9E9, 9E9, 9E9, 9E9, 9E9, 9E9]];
    CONST robtarget p12892:= [[1440.801902173912, -14.313092536989778, 1003.500033578516], [0, 0, 1, 0], [0, 0, 0, 0], [9E9, 9E9, 9E9, 9E9, 9E9, 9E9]];
    CONST robtarget p12893:= [[1440.6295674836624, -13.614108428227574, 1003.500033578516], [0, 0, 1, 0], [0, 0, 0, 0], [9E9, 9E9, 9E9, 9E9, 9E9, 9E9]];
    CONST robtarget p12894:= [[1440.5553749731691, -13.214334468469744, 1003.500033578516], [0, 0, 1, 0], [0, 0, 0, 0], [9E9, 9E9, 9E9, 9E9, 9E9, 9E9]];
    CONST robtarget p12895:= [[1440.4640328457035, -12.709422306143559, 1003.500033578516], [0, 0, 1, 0], [0, 0, 0, 0], [9E9, 9E9, 9E9, 9E9, 9E9, 9E9]];
    CONST robtarget p12896:= [[1440.3030274571006, -12.084967357370488, 1003.500033578516], [0, 0, 1, 0], [0, 0, 0, 0], [9E9, 9E9, 9E9, 9E9, 9E9, 9E9]];
    CONST robtarget p12897:= [[1440.1327454765292, -11.134713221206333, 1003.500033578516], [0, 0, 1, 0], [0, 0, 0, 0], [9E9, 9E9, 9E9, 9E9, 9E9, 9E9]];
    CONST robtarget p12898:= [[1440.082606622329, -10.835277709338492, 1003.500033578516], [0, 0, 1, 0], [0, 0, 0, 0], [9E9, 9E9, 9E9, 9E9, 9E9, 9E9]];
    CONST robtarget p12899:= [[1440.0250907351044, -10.515171219575677, 1003.500033578516], [0, 0, 1, 0], [0, 0, 0, 0], [9E9, 9E9, 9E9, 9E9, 9E9, 9E9]];
    CONST robtarget p12900:= [[1439.9964849308842, -10.317534875814047, 1003.500033578516], [0, 0, 1, 0], [0, 0, 0, 0], [9E9, 9E9, 9E9, 9E9, 9E9, 9E9]];
    CONST robtarget p12901:= [[1439.7942420605493, -9.237053558005769, 1003.500033578516], [0, 0, 1, 0], [0, 0, 0, 0], [9E9, 9E9, 9E9, 9E9, 9E9, 9E9]];
    CONST robtarget p12902:= [[1439.7517493771202, -9.0898646782763, 1003.500033578516], [0, 0, 1, 0], [0, 0, 0, 0], [9E9, 9E9, 9E9, 9E9, 9E9, 9E9]];
    CONST robtarget p12903:= [[1439.6740404066593, -8.474051703748337, 1003.500033578516], [0, 0, 1, 0], [0, 0, 0, 0], [9E9, 9E9, 9E9, 9E9, 9E9, 9E9]];
    CONST robtarget p12904:= [[1439.6348044276428, -8.175473894720803, 1003.500033578516], [0, 0, 1, 0], [0, 0, 0, 0], [9E9, 9E9, 9E9, 9E9, 9E9, 9E9]];
    CONST robtarget p12905:= [[1439.521959784018, -7.152764394782238, 1003.500033578516], [0, 0, 1, 0], [0, 0, 0, 0], [9E9, 9E9, 9E9, 9E9, 9E9, 9E9]];
    CONST robtarget p12906:= [[1439.5115214122834, -7.0320070770883305, 1003.500033578516], [0, 0, 1, 0], [0, 0, 0, 0], [9E9, 9E9, 9E9, 9E9, 9E9, 9E9]];
    CONST robtarget p12907:= [[1439.450635599965, -6.513422017207631, 1003.500033578516], [0, 0, 1, 0], [0, 0, 0, 0], [9E9, 9E9, 9E9, 9E9, 9E9, 9E9]];
    CONST robtarget p12908:= [[1439.3671769072694, -5.662637301603965, 1003.500033578516], [0, 0, 1, 0], [0, 0, 0, 0], [9E9, 9E9, 9E9, 9E9, 9E9, 9E9]];
    CONST robtarget p12909:= [[1439.2870375491386, -5.038098157890303, 1003.500033578516], [0, 0, 1, 0], [0, 0, 0, 0], [9E9, 9E9, 9E9, 9E9, 9E9, 9E9]];
    CONST robtarget p12910:= [[1439.2735725397006, -4.888813035853019, 1003.500033578516], [0, 0, 1, 0], [0, 0, 0, 0], [9E9, 9E9, 9E9, 9E9, 9E9, 9E9]];
    CONST robtarget p12911:= [[1439.2262678056295, -4.470426171482302, 1003.500033578516], [0, 0, 1, 0], [0, 0, 0, 0], [9E9, 9E9, 9E9, 9E9, 9E9, 9E9]];
    CONST robtarget p12912:= [[1439.2059324039976, -3.5753916485149517, 1003.500033578516], [0, 0, 1, 0], [0, 0, 0, 0], [9E9, 9E9, 9E9, 9E9, 9E9, 9E9]];
    CONST robtarget p12913:= [[1438.1672387091955, -2.9274487591431466, 1004.500033578516], [0, 0, 1, 0], [0, 0, 0, 0], [9E9, 9E9, 9E9, 9E9, 9E9, 9E9]];
    CONST robtarget p12914:= [[1438.1568657025232, -2.253387526526552, 1004.500033578516], [0, 0, 1, 0], [0, 0, 0, 0], [9E9, 9E9, 9E9, 9E9, 9E9, 9E9]];
    CONST robtarget p12915:= [[1438.1173308420125, -1.5040625307995583, 1004.500033578516], [0, 0, 1, 0], [0, 0, 0, 0], [9E9, 9E9, 9E9, 9E9, 9E9, 9E9]];
    CONST robtarget p12916:= [[1438.0954048626302, -1.15082460748431, 1004.500033578516], [0, 0, 1, 0], [0, 0, 0, 0], [9E9, 9E9, 9E9, 9E9, 9E9, 9E9]];
    CONST robtarget p12917:= [[1438.1060321975117, -0.8449536938244364, 1004.500033578516], [0, 0, 1, 0], [0, 0, 0, 0], [9E9, 9E9, 9E9, 9E9, 9E9, 9E9]];
    CONST robtarget p12918:= [[1438.1046446981748, -0.5846178324217135, 1004.500033578516], [0, 0, 1, 0], [0, 0, 0, 0], [9E9, 9E9, 9E9, 9E9, 9E9, 9E9]];
    CONST robtarget p12919:= [[1438.1039455215077, -0.13789397503474277, 1004.500033578516], [0, 0, 1, 0], [0, 0, 0, 0], [9E9, 9E9, 9E9, 9E9, 9E9, 9E9]];
    CONST robtarget p12920:= [[1438.0809624535589, 0.47733749171682405, 1004.500033578516], [0, 0, 1, 0], [0, 0, 0, 0], [9E9, 9E9, 9E9, 9E9, 9E9, 9E9]];
    CONST robtarget p12921:= [[1438.1046795365296, 1.2960851750493418, 1004.500033578516], [0, 0, 1, 0], [0, 0, 0, 0], [9E9, 9E9, 9E9, 9E9, 9E9, 9E9]];
    CONST robtarget p12922:= [[1438.1233916585004, 1.8355294746827013, 1004.500033578516], [0, 0, 1, 0], [0, 0, 0, 0], [9E9, 9E9, 9E9, 9E9, 9E9, 9E9]];
    CONST robtarget p12923:= [[1438.133347411806, 2.189769952394002, 1004.500033578516], [0, 0, 1, 0], [0, 0, 0, 0], [9E9, 9E9, 9E9, 9E9, 9E9, 9E9]];
    CONST robtarget p12924:= [[1438.2218182257252, 2.9345017757945726, 1004.500033578516], [0, 0, 1, 0], [0, 0, 0, 0], [9E9, 9E9, 9E9, 9E9, 9E9, 9E9]];
    CONST robtarget p12925:= [[1438.2240454410962, 3.5998157233707246, 1004.500033578516], [0, 0, 1, 0], [0, 0, 0, 0], [9E9, 9E9, 9E9, 9E9, 9E9, 9E9]];
    CONST robtarget p12926:= [[1438.2538525974223, 4.264485064438816, 1004.500033578516], [0, 0, 1, 0], [0, 0, 0, 0], [9E9, 9E9, 9E9, 9E9, 9E9, 9E9]];
    CONST robtarget p12927:= [[1438.2413712829468, 4.52593463232823, 1004.500033578516], [0, 0, 1, 0], [0, 0, 0, 0], [9E9, 9E9, 9E9, 9E9, 9E9, 9E9]];
    CONST robtarget p12928:= [[1438.289076178705, 5.023230440665756, 1004.500033578516], [0, 0, 1, 0], [0, 0, 0, 0], [9E9, 9E9, 9E9, 9E9, 9E9, 9E9]];
    CONST robtarget p12929:= [[1438.365900199651, 5.608795961981443, 1004.500033578516], [0, 0, 1, 0], [0, 0, 0, 0], [9E9, 9E9, 9E9, 9E9, 9E9, 9E9]];
    CONST robtarget p12930:= [[1438.3989350862762, 5.941241840837591, 1004.500033578516], [0, 0, 1, 0], [0, 0, 0, 0], [9E9, 9E9, 9E9, 9E9, 9E9, 9E9]];
    CONST robtarget p12931:= [[1438.4455119018257, 6.508953528354368, 1004.500033578516], [0, 0, 1, 0], [0, 0, 0, 0], [9E9, 9E9, 9E9, 9E9, 9E9, 9E9]];
    CONST robtarget p12932:= [[1438.5011309868592, 6.909521825300217, 1004.500033578516], [0, 0, 1, 0], [0, 0, 0, 0], [9E9, 9E9, 9E9, 9E9, 9E9, 9E9]];
    CONST robtarget p12933:= [[1438.5359799399607, 7.283167595526251, 1004.500033578516], [0, 0, 1, 0], [0, 0, 0, 0], [9E9, 9E9, 9E9, 9E9, 9E9, 9E9]];
    CONST robtarget p12934:= [[1438.5566577269171, 7.476140442983834, 1004.500033578516], [0, 0, 1, 0], [0, 0, 0, 0], [9E9, 9E9, 9E9, 9E9, 9E9, 9E9]];
    CONST robtarget p12935:= [[1438.6608200460387, 8.331317265199885, 1004.500033578516], [0, 0, 1, 0], [0, 0, 0, 0], [9E9, 9E9, 9E9, 9E9, 9E9, 9E9]];
    CONST robtarget p12936:= [[1438.6677466117833, 8.490785812525417, 1004.500033578516], [0, 0, 1, 0], [0, 0, 0, 0], [9E9, 9E9, 9E9, 9E9, 9E9, 9E9]];
    CONST robtarget p12937:= [[1438.6896854831043, 8.688290233967948, 1004.500033578516], [0, 0, 1, 0], [0, 0, 0, 0], [9E9, 9E9, 9E9, 9E9, 9E9, 9E9]];
    CONST robtarget p12938:= [[1438.744093940627, 9.041206100728871, 1004.500033578516], [0, 0, 1, 0], [0, 0, 0, 0], [9E9, 9E9, 9E9, 9E9, 9E9, 9E9]];
    CONST robtarget p12939:= [[1438.8391971414578, 9.637523042220195, 1004.500033578516], [0, 0, 1, 0], [0, 0, 0, 0], [9E9, 9E9, 9E9, 9E9, 9E9, 9E9]];
    CONST robtarget p12940:= [[1438.9646331271435, 10.125734554345087, 1004.500033578516], [0, 0, 1, 0], [0, 0, 0, 0], [9E9, 9E9, 9E9, 9E9, 9E9, 9E9]];
    CONST robtarget p12941:= [[1439.0536373750538, 10.756832810027419, 1004.500033578516], [0, 0, 1, 0], [0, 0, 0, 0], [9E9, 9E9, 9E9, 9E9, 9E9, 9E9]];
    CONST robtarget p12942:= [[1439.10801463163, 11.032032710785856, 1004.500033578516], [0, 0, 1, 0], [0, 0, 0, 0], [9E9, 9E9, 9E9, 9E9, 9E9, 9E9]];
    CONST robtarget p12943:= [[1439.1482117126516, 11.310126172200484, 1004.500033578516], [0, 0, 1, 0], [0, 0, 0, 0], [9E9, 9E9, 9E9, 9E9, 9E9, 9E9]];
    CONST robtarget p12944:= [[1439.1840746444127, 11.487491287232572, 1004.500033578516], [0, 0, 1, 0], [0, 0, 0, 0], [9E9, 9E9, 9E9, 9E9, 9E9, 9E9]];
    CONST robtarget p12945:= [[1439.2883629199086, 11.907972783981634, 1004.500033578516], [0, 0, 1, 0], [0, 0, 0, 0], [9E9, 9E9, 9E9, 9E9, 9E9, 9E9]];
    CONST robtarget p12946:= [[1439.4038535603247, 12.469502738683062, 1004.500033578516], [0, 0, 1, 0], [0, 0, 0, 0], [9E9, 9E9, 9E9, 9E9, 9E9, 9E9]];
    CONST robtarget p12947:= [[1439.59570790125, 13.66954299217052, 1004.500033578516], [0, 0, 1, 0], [0, 0, 0, 0], [9E9, 9E9, 9E9, 9E9, 9E9, 9E9]];
    CONST robtarget p12948:= [[1439.6662933490882, 13.925482700790965, 1004.500033578516], [0, 0, 1, 0], [0, 0, 0, 0], [9E9, 9E9, 9E9, 9E9, 9E9, 9E9]];
    CONST robtarget p12949:= [[1439.7764203897232, 14.32771265162431, 1004.500033578516], [0, 0, 1, 0], [0, 0, 0, 0], [9E9, 9E9, 9E9, 9E9, 9E9, 9E9]];
    CONST robtarget p12950:= [[1439.8456440272141, 14.627113374540954, 1004.500033578516], [0, 0, 1, 0], [0, 0, 0, 0], [9E9, 9E9, 9E9, 9E9, 9E9, 9E9]];
    CONST robtarget p12951:= [[1439.9781741742522, 15.152421312944284, 1004.500033578516], [0, 0, 1, 0], [0, 0, 0, 0], [9E9, 9E9, 9E9, 9E9, 9E9, 9E9]];
    CONST robtarget p12952:= [[1440.1037499954843, 15.540829390319743, 1004.500033578516], [0, 0, 1, 0], [0, 0, 0, 0], [9E9, 9E9, 9E9, 9E9, 9E9, 9E9]];
    CONST robtarget p12953:= [[1440.2679188270733, 16.118715091012447, 1004.500033578516], [0, 0, 1, 0], [0, 0, 0, 0], [9E9, 9E9, 9E9, 9E9, 9E9, 9E9]];
    CONST robtarget p12954:= [[1440.3518166725057, 16.58109319907109, 1004.500033578516], [0, 0, 1, 0], [0, 0, 0, 0], [9E9, 9E9, 9E9, 9E9, 9E9, 9E9]];
    CONST robtarget p12955:= [[1440.6391133588263, 17.552962261983524, 1004.500033578516], [0, 0, 1, 0], [0, 0, 0, 0], [9E9, 9E9, 9E9, 9E9, 9E9, 9E9]];
    CONST robtarget p12956:= [[1440.7040624992787, 17.88246122246754, 1004.500033578516], [0, 0, 1, 0], [0, 0, 0, 0], [9E9, 9E9, 9E9, 9E9, 9E9, 9E9]];
    CONST robtarget p12957:= [[1440.8038112315887, 18.1779549863669, 1004.500033578516], [0, 0, 1, 0], [0, 0, 0, 0], [9E9, 9E9, 9E9, 9E9, 9E9, 9E9]];
    CONST robtarget p12958:= [[1440.986288312718, 18.66708270849486, 1004.500033578516], [0, 0, 1, 0], [0, 0, 0, 0], [9E9, 9E9, 9E9, 9E9, 9E9, 9E9]];
    CONST robtarget p12959:= [[1441.272999809038, 19.500208001024845, 1004.500033578516], [0, 0, 1, 0], [0, 0, 0, 0], [9E9, 9E9, 9E9, 9E9, 9E9, 9E9]];
    CONST robtarget p12960:= [[1441.3774639679536, 19.8839614576046, 1004.500033578516], [0, 0, 1, 0], [0, 0, 0, 0], [9E9, 9E9, 9E9, 9E9, 9E9, 9E9]];
    CONST robtarget p12961:= [[1441.5989839532842, 20.493133960258263, 1004.500033578516], [0, 0, 1, 0], [0, 0, 0, 0], [9E9, 9E9, 9E9, 9E9, 9E9, 9E9]];
    CONST robtarget p12962:= [[1441.872508477147, 21.299335752536166, 1004.500033578516], [0, 0, 1, 0], [0, 0, 0, 0], [9E9, 9E9, 9E9, 9E9, 9E9, 9E9]];
    CONST robtarget p12963:= [[1442.2084045943604, 22.285469150960267, 1004.500033578516], [0, 0, 1, 0], [0, 0, 0, 0], [9E9, 9E9, 9E9, 9E9, 9E9, 9E9]];
    CONST robtarget p12964:= [[1442.3792051158814, 22.679146625628732, 1004.500033578516], [0, 0, 1, 0], [0, 0, 0, 0], [9E9, 9E9, 9E9, 9E9, 9E9, 9E9]];
    CONST robtarget p12965:= [[1442.6374114637401, 23.294422849661572, 1004.500033578516], [0, 0, 1, 0], [0, 0, 0, 0], [9E9, 9E9, 9E9, 9E9, 9E9, 9E9]];
    CONST robtarget p12966:= [[1442.9574489919146, 24.046927460017628, 1004.500033578516], [0, 0, 1, 0], [0, 0, 0, 0], [9E9, 9E9, 9E9, 9E9, 9E9, 9E9]];
    CONST robtarget p12967:= [[1443.3020407335125, 24.857238852462316, 1004.500033578516], [0, 0, 1, 0], [0, 0, 0, 0], [9E9, 9E9, 9E9, 9E9, 9E9, 9E9]];
    CONST robtarget p12968:= [[1443.597267180258, 25.47780754694601, 1004.500033578516], [0, 0, 1, 0], [0, 0, 0, 0], [9E9, 9E9, 9E9, 9E9, 9E9, 9E9]];
    CONST robtarget p12969:= [[1443.6518649466536, 25.583889591562397, 1004.500033578516], [0, 0, 1, 0], [0, 0, 0, 0], [9E9, 9E9, 9E9, 9E9, 9E9, 9E9]];
    CONST robtarget p12970:= [[1443.9563563177499, 26.23189734339482, 1004.500033578516], [0, 0, 1, 0], [0, 0, 0, 0], [9E9, 9E9, 9E9, 9E9, 9E9, 9E9]];
    CONST robtarget p12971:= [[1444.169960455085, 26.761050425769028, 1004.500033578516], [0, 0, 1, 0], [0, 0, 0, 0], [9E9, 9E9, 9E9, 9E9, 9E9, 9E9]];
    CONST robtarget p12972:= [[1444.2434165844604, 26.93826578144443, 1004.500033578516], [0, 0, 1, 0], [0, 0, 0, 0], [9E9, 9E9, 9E9, 9E9, 9E9, 9E9]];
    CONST robtarget p12973:= [[1444.3705175144653, 27.175502336913524, 1004.500033578516], [0, 0, 1, 0], [0, 0, 0, 0], [9E9, 9E9, 9E9, 9E9, 9E9, 9E9]];
    CONST robtarget p12974:= [[1444.6748368555316, 27.765408547356856, 1004.500033578516], [0, 0, 1, 0], [0, 0, 0, 0], [9E9, 9E9, 9E9, 9E9, 9E9, 9E9]];
    CONST robtarget p12975:= [[1444.9084378894538, 28.197308708981268, 1004.500033578516], [0, 0, 1, 0], [0, 0, 0, 0], [9E9, 9E9, 9E9, 9E9, 9E9, 9E9]];
    CONST robtarget p12976:= [[1445.1818052066146, 28.70127785739271, 1004.500033578516], [0, 0, 1, 0], [0, 0, 0, 0], [9E9, 9E9, 9E9, 9E9, 9E9, 9E9]];
    CONST robtarget p12977:= [[1445.4944762899863, 29.34583193673508, 1004.500033578516], [0, 0, 1, 0], [0, 0, 0, 0], [9E9, 9E9, 9E9, 9E9, 9E9, 9E9]];
    CONST robtarget p12978:= [[1445.7261447752903, 29.814330618031804, 1004.500033578516], [0, 0, 1, 0], [0, 0, 0, 0], [9E9, 9E9, 9E9, 9E9, 9E9, 9E9]];
    CONST robtarget p12979:= [[1445.973531868932, 30.288426423587893, 1004.500033578516], [0, 0, 1, 0], [0, 0, 0, 0], [9E9, 9E9, 9E9, 9E9, 9E9, 9E9]];
    CONST robtarget p12980:= [[1446.2950487789296, 30.827622416643536, 1004.500033578516], [0, 0, 1, 0], [0, 0, 0, 0], [9E9, 9E9, 9E9, 9E9, 9E9, 9E9]];
    CONST robtarget p12981:= [[1446.553405291924, 31.224459687935024, 1004.500033578516], [0, 0, 1, 0], [0, 0, 0, 0], [9E9, 9E9, 9E9, 9E9, 9E9, 9E9]];
    CONST robtarget p12982:= [[1446.8826655319328, 31.742105921892957, 1004.500033578516], [0, 0, 1, 0], [0, 0, 0, 0], [9E9, 9E9, 9E9, 9E9, 9E9, 9E9]];
    CONST robtarget p12983:= [[1447.19537451066, 32.228981845091724, 1004.500033578516], [0, 0, 1, 0], [0, 0, 0, 0], [9E9, 9E9, 9E9, 9E9, 9E9, 9E9]];
    CONST robtarget p12984:= [[1447.475572177372, 32.75800709336238, 1004.500033578516], [0, 0, 1, 0], [0, 0, 0, 0], [9E9, 9E9, 9E9, 9E9, 9E9, 9E9]];
    CONST robtarget p12985:= [[1447.6044411484218, 32.97092323237857, 1004.500033578516], [0, 0, 1, 0], [0, 0, 0, 0], [9E9, 9E9, 9E9, 9E9, 9E9, 9E9]];
    CONST robtarget p12986:= [[1447.7348260477963, 33.1773299437759, 1004.500033578516], [0, 0, 1, 0], [0, 0, 0, 0], [9E9, 9E9, 9E9, 9E9, 9E9, 9E9]];
    CONST robtarget p12987:= [[1447.9475189252498, 33.53243863646705, 1004.500033578516], [0, 0, 1, 0], [0, 0, 0, 0], [9E9, 9E9, 9E9, 9E9, 9E9, 9E9]];
    CONST robtarget p12988:= [[1448.3956378006717, 34.23661589228632, 1004.500033578516], [0, 0, 1, 0], [0, 0, 0, 0], [9E9, 9E9, 9E9, 9E9, 9E9, 9E9]];
    CONST robtarget p12989:= [[1448.5981810801766, 34.52770354434266, 1004.500033578516], [0, 0, 1, 0], [0, 0, 0, 0], [9E9, 9E9, 9E9, 9E9, 9E9, 9E9]];
    CONST robtarget p12990:= [[1448.8190030731525, 34.814548628749435, 1004.500033578516], [0, 0, 1, 0], [0, 0, 0, 0], [9E9, 9E9, 9E9, 9E9, 9E9, 9E9]];
    CONST robtarget p12991:= [[1449.2669476690887, 35.47367328000813, 1004.500033578516], [0, 0, 1, 0], [0, 0, 0, 0], [9E9, 9E9, 9E9, 9E9, 9E9, 9E9]];
    CONST robtarget p12992:= [[1449.3877570230256, 35.638578685967275, 1004.500033578516], [0, 0, 1, 0], [0, 0, 0, 0], [9E9, 9E9, 9E9, 9E9, 9E9, 9E9]];
    CONST robtarget p12993:= [[1449.900683771793, 36.305431331343385, 1004.500033578516], [0, 0, 1, 0], [0, 0, 0, 0], [9E9, 9E9, 9E9, 9E9, 9E9, 9E9]];
    CONST robtarget p12994:= [[1450.1516072887596, 36.649397047990405, 1004.500033578516], [0, 0, 1, 0], [0, 0, 0, 0], [9E9, 9E9, 9E9, 9E9, 9E9, 9E9]];
    CONST robtarget p12995:= [[1450.596295568302, 37.337110189375, 1004.500033578516], [0, 0, 1, 0], [0, 0, 0, 0], [9E9, 9E9, 9E9, 9E9, 9E9, 9E9]];
    CONST robtarget p12996:= [[1450.900796772915, 37.758546405141374, 1004.500033578516], [0, 0, 1, 0], [0, 0, 0, 0], [9E9, 9E9, 9E9, 9E9, 9E9, 9E9]];
    CONST robtarget p12997:= [[1451.005491734291, 37.87992358758659, 1004.500033578516], [0, 0, 1, 0], [0, 0, 0, 0], [9E9, 9E9, 9E9, 9E9, 9E9, 9E9]];
    CONST robtarget p12998:= [[1451.1585381103691, 38.070759027472306, 1004.500033578516], [0, 0, 1, 0], [0, 0, 0, 0], [9E9, 9E9, 9E9, 9E9, 9E9, 9E9]];
    CONST robtarget p12999:= [[1451.5310829838745, 38.493064738246204, 1004.500033578516], [0, 0, 1, 0], [0, 0, 0, 0], [9E9, 9E9, 9E9, 9E9, 9E9, 9E9]];
    CONST robtarget p13000:= [[1451.695332903664, 38.68895195446778, 1004.500033578516], [0, 0, 1, 0], [0, 0, 0, 0], [9E9, 9E9, 9E9, 9E9, 9E9, 9E9]];
    CONST robtarget p13001:= [[1452.2777833465054, 39.37606287256422, 1004.500033578516], [0, 0, 1, 0], [0, 0, 0, 0], [9E9, 9E9, 9E9, 9E9, 9E9, 9E9]];
    CONST robtarget p13002:= [[1452.7004845231236, 39.90931303978361, 1004.500033578516], [0, 0, 1, 0], [0, 0, 0, 0], [9E9, 9E9, 9E9, 9E9, 9E9, 9E9]];
    CONST robtarget p13003:= [[1452.842140429859, 40.108093010893896, 1004.500033578516], [0, 0, 1, 0], [0, 0, 0, 0], [9E9, 9E9, 9E9, 9E9, 9E9, 9E9]];
    CONST robtarget p13004:= [[1453.06171089215, 40.34580318158747, 1004.500033578516], [0, 0, 1, 0], [0, 0, 0, 0], [9E9, 9E9, 9E9, 9E9, 9E9, 9E9]];
    CONST robtarget p13005:= [[1453.088979517739, 40.3733326620529, 1004.500033578516], [0, 0, 1, 0], [0, 0, 0, 0], [9E9, 9E9, 9E9, 9E9, 9E9, 9E9]];
    CONST robtarget p13006:= [[1453.6502318219732, 41.04645579317399, 1004.500033578516], [0, 0, 1, 0], [0, 0, 0, 0], [9E9, 9E9, 9E9, 9E9, 9E9, 9E9]];
    CONST robtarget p13007:= [[1453.9387433825884, 41.35256729943596, 1004.500033578516], [0, 0, 1, 0], [0, 0, 0, 0], [9E9, 9E9, 9E9, 9E9, 9E9, 9E9]];
    CONST robtarget p13008:= [[1454.0974802012552, 41.54009858812887, 1004.500033578516], [0, 0, 1, 0], [0, 0, 0, 0], [9E9, 9E9, 9E9, 9E9, 9E9, 9E9]];
    CONST robtarget p13009:= [[1454.386096339884, 41.869725401464535, 1004.500033578516], [0, 0, 1, 0], [0, 0, 0, 0], [9E9, 9E9, 9E9, 9E9, 9E9, 9E9]];
    CONST robtarget p13010:= [[1454.9990611769722, 42.501629511381935, 1004.500033578516], [0, 0, 1, 0], [0, 0, 0, 0], [9E9, 9E9, 9E9, 9E9, 9E9, 9E9]];
    CONST robtarget p13011:= [[1455.4936645154014, 42.995984938290846, 1004.500033578516], [0, 0, 1, 0], [0, 0, 0, 0], [9E9, 9E9, 9E9, 9E9, 9E9, 9E9]];
    CONST robtarget p13012:= [[1456.0558922076536, 43.60967233657556, 1004.500033578516], [0, 0, 1, 0], [0, 0, 0, 0], [9E9, 9E9, 9E9, 9E9, 9E9, 9E9]];
    CONST robtarget p13013:= [[1456.5187328460422, 44.068238199093145, 1004.500033578516], [0, 0, 1, 0], [0, 0, 0, 0], [9E9, 9E9, 9E9, 9E9, 9E9, 9E9]];
    CONST robtarget p13014:= [[1456.8456377622501, 44.37271094491153, 1004.500033578516], [0, 0, 1, 0], [0, 0, 0, 0], [9E9, 9E9, 9E9, 9E9, 9E9, 9E9]];
    CONST robtarget p13015:= [[1457.2451057007893, 44.780465272619466, 1004.500033578516], [0, 0, 1, 0], [0, 0, 0, 0], [9E9, 9E9, 9E9, 9E9, 9E9, 9E9]];
    CONST robtarget p13016:= [[1457.9609854160976, 45.438676793561484, 1004.500033578516], [0, 0, 1, 0], [0, 0, 0, 0], [9E9, 9E9, 9E9, 9E9, 9E9, 9E9]];
    CONST robtarget p13017:= [[1458.2152632374716, 45.67130715052407, 1004.500033578516], [0, 0, 1, 0], [0, 0, 0, 0], [9E9, 9E9, 9E9, 9E9, 9E9, 9E9]];
    CONST robtarget p13018:= [[1458.4510864758895, 45.879986281072476, 1004.500033578516], [0, 0, 1, 0], [0, 0, 0, 0], [9E9, 9E9, 9E9, 9E9, 9E9, 9E9]];
    CONST robtarget p13019:= [[1458.9635156809188, 46.287722618122345, 1004.500033578516], [0, 0, 1, 0], [0, 0, 0, 0], [9E9, 9E9, 9E9, 9E9, 9E9, 9E9]];
    CONST robtarget p13020:= [[1459.2531765279584, 46.521135733037326, 1004.500033578516], [0, 0, 1, 0], [0, 0, 0, 0], [9E9, 9E9, 9E9, 9E9, 9E9, 9E9]];
    CONST robtarget p13021:= [[1459.502874391438, 46.74271746704248, 1004.500033578516], [0, 0, 1, 0], [0, 0, 0, 0], [9E9, 9E9, 9E9, 9E9, 9E9, 9E9]];
    CONST robtarget p13022:= [[1459.8253100070629, 47.037729172734956, 1004.500033578516], [0, 0, 1, 0], [0, 0, 0, 0], [9E9, 9E9, 9E9, 9E9, 9E9, 9E9]];
    CONST robtarget p13023:= [[1460.1833773690096, 47.382085392396476, 1004.500033578516], [0, 0, 1, 0], [0, 0, 0, 0], [9E9, 9E9, 9E9, 9E9, 9E9, 9E9]];
    CONST robtarget p13024:= [[1460.643450662835, 47.801816748479126, 1004.500033578516], [0, 0, 1, 0], [0, 0, 0, 0], [9E9, 9E9, 9E9, 9E9, 9E9, 9E9]];
    CONST robtarget p13025:= [[1460.8077304131712, 47.91834774655288, 1004.500033578516], [0, 0, 1, 0], [0, 0, 0, 0], [9E9, 9E9, 9E9, 9E9, 9E9, 9E9]];
    CONST robtarget p13026:= [[1461.326709579753, 48.327508639145364, 1004.500033578516], [0, 0, 1, 0], [0, 0, 0, 0], [9E9, 9E9, 9E9, 9E9, 9E9, 9E9]];
    CONST robtarget p13027:= [[1461.5674134886187, 48.50766899539698, 1004.500033578516], [0, 0, 1, 0], [0, 0, 0, 0], [9E9, 9E9, 9E9, 9E9, 9E9, 9E9]];
    CONST robtarget p13028:= [[1462.0494276242036, 48.88193797292574, 1004.500033578516], [0, 0, 1, 0], [0, 0, 0, 0], [9E9, 9E9, 9E9, 9E9, 9E9, 9E9]];
    CONST robtarget p13029:= [[1462.624800249608, 49.3185130840026, 1004.500033578516], [0, 0, 1, 0], [0, 0, 0, 0], [9E9, 9E9, 9E9, 9E9, 9E9, 9E9]];
    CONST robtarget p13030:= [[1462.9086209744496, 49.546691234083625, 1004.500033578516], [0, 0, 1, 0], [0, 0, 0, 0], [9E9, 9E9, 9E9, 9E9, 9E9, 9E9]];
    CONST robtarget p13031:= [[1463.4413467535194, 49.97852336366911, 1004.500033578516], [0, 0, 1, 0], [0, 0, 0, 0], [9E9, 9E9, 9E9, 9E9, 9E9, 9E9]];
    CONST robtarget p13032:= [[1463.537736242698, 50.04063540955296, 1004.500033578516], [0, 0, 1, 0], [0, 0, 0, 0], [9E9, 9E9, 9E9, 9E9, 9E9, 9E9]];
    CONST robtarget p13033:= [[1464.2626033115732, 50.55465159390842, 1004.500033578516], [0, 0, 1, 0], [0, 0, 0, 0], [9E9, 9E9, 9E9, 9E9, 9E9, 9E9]];
    CONST robtarget p13034:= [[1464.4516006526624, 50.70078681042875, 1004.500033578516], [0, 0, 1, 0], [0, 0, 0, 0], [9E9, 9E9, 9E9, 9E9, 9E9, 9E9]];
    CONST robtarget p13035:= [[1464.6450121186099, 50.81474515054116, 1004.500033578516], [0, 0, 1, 0], [0, 0, 0, 0], [9E9, 9E9, 9E9, 9E9, 9E9, 9E9]];
    CONST robtarget p13036:= [[1464.9842238382282, 51.041152846211844, 1004.500033578516], [0, 0, 1, 0], [0, 0, 0, 0], [9E9, 9E9, 9E9, 9E9, 9E9, 9E9]];
    CONST robtarget p13037:= [[1465.2966890025812, 51.24541736495463, 1004.500033578516], [0, 0, 1, 0], [0, 0, 0, 0], [9E9, 9E9, 9E9, 9E9, 9E9, 9E9]];
    CONST robtarget p13038:= [[1465.7784670109545, 51.57449702888138, 1004.500033578516], [0, 0, 1, 0], [0, 0, 0, 0], [9E9, 9E9, 9E9, 9E9, 9E9, 9E9]];
    CONST robtarget p13039:= [[1466.4583565838625, 51.99071500357397, 1004.500033578516], [0, 0, 1, 0], [0, 0, 0, 0], [9E9, 9E9, 9E9, 9E9, 9E9, 9E9]];
    CONST robtarget p13040:= [[1466.897742208927, 52.301957908302924, 1004.500033578516], [0, 0, 1, 0], [0, 0, 0, 0], [9E9, 9E9, 9E9, 9E9, 9E9, 9E9]];
    CONST robtarget p13041:= [[1467.3453131395365, 52.620184186844014, 1004.500033578516], [0, 0, 1, 0], [0, 0, 0, 0], [9E9, 9E9, 9E9, 9E9, 9E9, 9E9]];
    CONST robtarget p13042:= [[1467.7138756141005, 52.84703896959475, 1004.500033578516], [0, 0, 1, 0], [0, 0, 0, 0], [9E9, 9E9, 9E9, 9E9, 9E9, 9E9]];
    CONST robtarget p13043:= [[1467.7635266520087, 52.87332950926053, 1004.500033578516], [0, 0, 1, 0], [0, 0, 0, 0], [9E9, 9E9, 9E9, 9E9, 9E9, 9E9]];
    CONST robtarget p13044:= [[1468.1652901881937, 53.082614180834426, 1004.500033578516], [0, 0, 1, 0], [0, 0, 0, 0], [9E9, 9E9, 9E9, 9E9, 9E9, 9E9]];
    CONST robtarget p13045:= [[1468.4567539152058, 53.25022355346029, 1004.500033578516], [0, 0, 1, 0], [0, 0, 0, 0], [9E9, 9E9, 9E9, 9E9, 9E9, 9E9]];
    CONST robtarget p13046:= [[1468.872081059277, 53.4825532090569, 1004.500033578516], [0, 0, 1, 0], [0, 0, 0, 0], [9E9, 9E9, 9E9, 9E9, 9E9, 9E9]];
    CONST robtarget p13047:= [[1469.440127291126, 53.81975824631908, 1004.500033578516], [0, 0, 1, 0], [0, 0, 0, 0], [9E9, 9E9, 9E9, 9E9, 9E9, 9E9]];
    CONST robtarget p13048:= [[1469.5152781957622, 53.85887253191237, 1004.500033578516], [0, 0, 1, 0], [0, 0, 0, 0], [9E9, 9E9, 9E9, 9E9, 9E9, 9E9]];
    CONST robtarget p13049:= [[1470.3090029522718, 54.321846030326085, 1004.500033578516], [0, 0, 1, 0], [0, 0, 0, 0], [9E9, 9E9, 9E9, 9E9, 9E9, 9E9]];
    CONST robtarget p13050:= [[1470.6426378605752, 54.49383800588359, 1004.500033578516], [0, 0, 1, 0], [0, 0, 0, 0], [9E9, 9E9, 9E9, 9E9, 9E9, 9E9]];
    CONST robtarget p13051:= [[1470.9624417912746, 54.67422208195656, 1004.500033578516], [0, 0, 1, 0], [0, 0, 0, 0], [9E9, 9E9, 9E9, 9E9, 9E9, 9E9]];
    CONST robtarget p13052:= [[1471.4290172095116, 54.917236703203585, 1004.500033578516], [0, 0, 1, 0], [0, 0, 0, 0], [9E9, 9E9, 9E9, 9E9, 9E9, 9E9]];
    CONST robtarget p13053:= [[1471.5919616120848, 55.00960374657683, 1004.500033578516], [0, 0, 1, 0], [0, 0, 0, 0], [9E9, 9E9, 9E9, 9E9, 9E9, 9E9]];
    CONST robtarget p13054:= [[1471.991481448302, 55.199745091221274, 1004.500033578516], [0, 0, 1, 0], [0, 0, 0, 0], [9E9, 9E9, 9E9, 9E9, 9E9, 9E9]];
    CONST robtarget p13055:= [[1472.3620789232887, 55.392755390965945, 1004.500033578516], [0, 0, 1, 0], [0, 0, 0, 0], [9E9, 9E9, 9E9, 9E9, 9E9, 9E9]];
    CONST robtarget p13056:= [[1472.8871506814503, 55.65508946347448, 1004.500033578516], [0, 0, 1, 0], [0, 0, 0, 0], [9E9, 9E9, 9E9, 9E9, 9E9, 9E9]];
    CONST robtarget p13057:= [[1473.300801899863, 55.807576052207466, 1004.500033578516], [0, 0, 1, 0], [0, 0, 0, 0], [9E9, 9E9, 9E9, 9E9, 9E9, 9E9]];
    CONST robtarget p13058:= [[1474.160472529876, 56.23629796164731, 1004.500033578516], [0, 0, 1, 0], [0, 0, 0, 0], [9E9, 9E9, 9E9, 9E9, 9E9, 9E9]];
    CONST robtarget p13059:= [[1474.8757436771214, 56.58565627460129, 1004.500033578516], [0, 0, 1, 0], [0, 0, 0, 0], [9E9, 9E9, 9E9, 9E9, 9E9, 9E9]];
    CONST robtarget p13060:= [[1475.1700229552278, 56.72494849928697, 1004.500033578516], [0, 0, 1, 0], [0, 0, 0, 0], [9E9, 9E9, 9E9, 9E9, 9E9, 9E9]];
    CONST robtarget p13061:= [[1475.7376606289886, 56.96993125548407, 1004.500033578516], [0, 0, 1, 0], [0, 0, 0, 0], [9E9, 9E9, 9E9, 9E9, 9E9, 9E9]];
    CONST robtarget p13062:= [[1475.9102266338534, 57.03414733371747, 1004.500033578516], [0, 0, 1, 0], [0, 0, 0, 0], [9E9, 9E9, 9E9, 9E9, 9E9, 9E9]];
    CONST robtarget p13063:= [[1476.8606321214595, 57.421963337572194, 1004.500033578516], [0, 0, 1, 0], [0, 0, 0, 0], [9E9, 9E9, 9E9, 9E9, 9E9, 9E9]];
    CONST robtarget p13064:= [[1477.1388643936994, 57.50916375107862, 1004.500033578516], [0, 0, 1, 0], [0, 0, 0, 0], [9E9, 9E9, 9E9, 9E9, 9E9, 9E9]];
    CONST robtarget p13065:= [[1477.8663814157512, 57.80251877234741, 1004.500033578516], [0, 0, 1, 0], [0, 0, 0, 0], [9E9, 9E9, 9E9, 9E9, 9E9, 9E9]];
    CONST robtarget p13066:= [[1478.5401996156954, 58.06194508624084, 1004.500033578516], [0, 0, 1, 0], [0, 0, 0, 0], [9E9, 9E9, 9E9, 9E9, 9E9, 9E9]];
    CONST robtarget p13067:= [[1478.5955624902124, 58.08193091289037, 1004.500033578516], [0, 0, 1, 0], [0, 0, 0, 0], [9E9, 9E9, 9E9, 9E9, 9E9, 9E9]];
    CONST robtarget p13068:= [[1479.380133702607, 58.38084761341982, 1004.500033578516], [0, 0, 1, 0], [0, 0, 0, 0], [9E9, 9E9, 9E9, 9E9, 9E9, 9E9]];
    CONST robtarget p13069:= [[1479.6346720373388, 58.45865335615595, 1004.500033578516], [0, 0, 1, 0], [0, 0, 0, 0], [9E9, 9E9, 9E9, 9E9, 9E9, 9E9]];
    CONST robtarget p13070:= [[1480.281144256426, 58.69798114111386, 1004.500033578516], [0, 0, 1, 0], [0, 0, 0, 0], [9E9, 9E9, 9E9, 9E9, 9E9, 9E9]];
    CONST robtarget p13071:= [[1480.722858571609, 58.806307378157484, 1004.500033578516], [0, 0, 1, 0], [0, 0, 0, 0], [9E9, 9E9, 9E9, 9E9, 9E9, 9E9]];
    CONST robtarget p13072:= [[1481.2305072276276, 58.96031035587556, 1004.500033578516], [0, 0, 1, 0], [0, 0, 0, 0], [9E9, 9E9, 9E9, 9E9, 9E9, 9E9]];
    CONST robtarget p13073:= [[1481.8080426358185, 59.15153136180062, 1004.500033578516], [0, 0, 1, 0], [0, 0, 0, 0], [9E9, 9E9, 9E9, 9E9, 9E9, 9E9]];
    CONST robtarget p13074:= [[1482.4896986903746, 59.339320451982346, 1004.500033578516], [0, 0, 1, 0], [0, 0, 0, 0], [9E9, 9E9, 9E9, 9E9, 9E9, 9E9]];
    CONST robtarget p13075:= [[1483.4836216295314, 59.650399819698734, 1004.500033578516], [0, 0, 1, 0], [0, 0, 0, 0], [9E9, 9E9, 9E9, 9E9, 9E9, 9E9]];
    CONST robtarget p13076:= [[1483.7279088307253, 59.70000140214158, 1004.500033578516], [0, 0, 1, 0], [0, 0, 0, 0], [9E9, 9E9, 9E9, 9E9, 9E9, 9E9]];
    CONST robtarget p13077:= [[1484.3903358801856, 59.898374550917524, 1004.500033578516], [0, 0, 1, 0], [0, 0, 0, 0], [9E9, 9E9, 9E9, 9E9, 9E9, 9E9]];
    CONST robtarget p13078:= [[1484.9295411546261, 60.037303277865746, 1004.500033578516], [0, 0, 1, 0], [0, 0, 0, 0], [9E9, 9E9, 9E9, 9E9, 9E9, 9E9]];
    CONST robtarget p13079:= [[1485.4822955514733, 60.17132516748278, 1004.500033578516], [0, 0, 1, 0], [0, 0, 0, 0], [9E9, 9E9, 9E9, 9E9, 9E9, 9E9]];
    CONST robtarget p13080:= [[1485.83985165664, 60.26149444224349, 1004.500033578516], [0, 0, 1, 0], [0, 0, 0, 0], [9E9, 9E9, 9E9, 9E9, 9E9, 9E9]];
    CONST robtarget p13081:= [[1486.1725717214188, 60.33336224684079, 1004.500033578516], [0, 0, 1, 0], [0, 0, 0, 0], [9E9, 9E9, 9E9, 9E9, 9E9, 9E9]];
    CONST robtarget p13082:= [[1486.4035998328716, 60.3744819640696, 1004.500033578516], [0, 0, 1, 0], [0, 0, 0, 0], [9E9, 9E9, 9E9, 9E9, 9E9, 9E9]];
    CONST robtarget p13083:= [[1486.980620135331, 60.50822435451455, 1004.500033578516], [0, 0, 1, 0], [0, 0, 0, 0], [9E9, 9E9, 9E9, 9E9, 9E9, 9E9]];
    CONST robtarget p13084:= [[1487.2589365439774, 60.55520710476277, 1004.500033578516], [0, 0, 1, 0], [0, 0, 0, 0], [9E9, 9E9, 9E9, 9E9, 9E9, 9E9]];
    CONST robtarget p13085:= [[1488.2799587231377, 60.7973902374507, 1004.500033578516], [0, 0, 1, 0], [0, 0, 0, 0], [9E9, 9E9, 9E9, 9E9, 9E9, 9E9]];
    CONST robtarget p13086:= [[1488.955553570077, 60.941974607030275, 1004.500033578516], [0, 0, 1, 0], [0, 0, 0, 0], [9E9, 9E9, 9E9, 9E9, 9E9, 9E9]];
    CONST robtarget p13087:= [[1489.9483044159201, 61.04981764067968, 1004.500033578516], [0, 0, 1, 0], [0, 0, 0, 0], [9E9, 9E9, 9E9, 9E9, 9E9, 9E9]];
    CONST robtarget p13088:= [[1490.3277981435774, 61.11092543799903, 1004.500033578516], [0, 0, 1, 0], [0, 0, 0, 0], [9E9, 9E9, 9E9, 9E9, 9E9, 9E9]];
    CONST robtarget p13089:= [[1490.774155528875, 61.20961701565578, 1004.500033578516], [0, 0, 1, 0], [0, 0, 0, 0], [9E9, 9E9, 9E9, 9E9, 9E9, 9E9]];
    CONST robtarget p13090:= [[1491.7111391655485, 61.33687427489265, 1004.500033578516], [0, 0, 1, 0], [0, 0, 0, 0], [9E9, 9E9, 9E9, 9E9, 9E9, 9E9]];
    CONST robtarget p13091:= [[1491.8176109429833, 61.35539390702611, 1004.500033578516], [0, 0, 1, 0], [0, 0, 0, 0], [9E9, 9E9, 9E9, 9E9, 9E9, 9E9]];
    CONST robtarget p13092:= [[1492.7773147595299, 61.48804351914917, 1004.500033578516], [0, 0, 1, 0], [0, 0, 0, 0], [9E9, 9E9, 9E9, 9E9, 9E9, 9E9]];
    CONST robtarget p13093:= [[1493.3840917318282, 61.521590332794815, 1004.500033578516], [0, 0, 1, 0], [0, 0, 0, 0], [9E9, 9E9, 9E9, 9E9, 9E9, 9E9]];
    CONST robtarget p13094:= [[1494.4270587730696, 61.59652175427327, 1004.500033578516], [0, 0, 1, 0], [0, 0, 0, 0], [9E9, 9E9, 9E9, 9E9, 9E9, 9E9]];
    CONST robtarget p13095:= [[1495.131286778597, 61.68136149807346, 1004.500033578516], [0, 0, 1, 0], [0, 0, 0, 0], [9E9, 9E9, 9E9, 9E9, 9E9, 9E9]];
    CONST robtarget p13096:= [[1495.5364916097835, 61.73377876506605, 1004.500033578516], [0, 0, 1, 0], [0, 0, 0, 0], [9E9, 9E9, 9E9, 9E9, 9E9, 9E9]];
    CONST robtarget p13097:= [[1496.1515703316495, 61.782099586864106, 1004.500033578516], [0, 0, 1, 0], [0, 0, 0, 0], [9E9, 9E9, 9E9, 9E9, 9E9, 9E9]];
    CONST robtarget p13098:= [[1496.422447279113, 61.801413691535444, 1004.500033578516], [0, 0, 1, 0], [0, 0, 0, 0], [9E9, 9E9, 9E9, 9E9, 9E9, 9E9]];
    CONST robtarget p13099:= [[1497.6786265378842, 61.86040397479884, 1004.500033578516], [0, 0, 1, 0], [0, 0, 0, 0], [9E9, 9E9, 9E9, 9E9, 9E9, 9E9]];
    CONST robtarget p13100:= [[1498.1750717722493, 61.895311005823274, 1004.500033578516], [0, 0, 1, 0], [0, 0, 0, 0], [9E9, 9E9, 9E9, 9E9, 9E9, 9E9]];
    CONST robtarget p13101:= [[1499.009502160973, 61.89408246817733, 1004.500033578516], [0, 0, 1, 0], [0, 0, 0, 0], [9E9, 9E9, 9E9, 9E9, 9E9, 9E9]];
    CONST robtarget p13102:= [[1500.0126360978675, 61.883842619010025, 1004.500033578516], [0, 0, 1, 0], [0, 0, 0, 0], [9E9, 9E9, 9E9, 9E9, 9E9, 9E9]];
    CONST robtarget p13103:= [[1501.2639236069538, 61.87661928517919, 1004.500033578516], [0, 0, 1, 0], [0, 0, 0, 0], [9E9, 9E9, 9E9, 9E9, 9E9, 9E9]];
    CONST robtarget p13104:= [[1501.5748546373954, 61.88172748782357, 1004.500033578516], [0, 0, 1, 0], [0, 0, 0, 0], [9E9, 9E9, 9E9, 9E9, 9E9, 9E9]];
    CONST robtarget p13105:= [[1502.3446247528454, 61.86933119568256, 1004.500033578516], [0, 0, 1, 0], [0, 0, 0, 0], [9E9, 9E9, 9E9, 9E9, 9E9, 9E9]];
    CONST robtarget p13106:= [[1502.839149976785, 61.841160583035915, 1004.500033578516], [0, 0, 1, 0], [0, 0, 0, 0], [9E9, 9E9, 9E9, 9E9, 9E9, 9E9]];
    CONST robtarget p13107:= [[1503.5146996063968, 61.79321851483671, 1004.500033578516], [0, 0, 1, 0], [0, 0, 0, 0], [9E9, 9E9, 9E9, 9E9, 9E9, 9E9]];
    CONST robtarget p13108:= [[1503.81567358534, 61.77831064618785, 1004.500033578516], [0, 0, 1, 0], [0, 0, 0, 0], [9E9, 9E9, 9E9, 9E9, 9E9, 9E9]];
    CONST robtarget p13109:= [[1504.7228555992383, 61.70277962853193, 1004.500033578516], [0, 0, 1, 0], [0, 0, 0, 0], [9E9, 9E9, 9E9, 9E9, 9E9, 9E9]];
    CONST robtarget p13110:= [[1504.9515836673077, 61.66633742969158, 1004.500033578516], [0, 0, 1, 0], [0, 0, 0, 0], [9E9, 9E9, 9E9, 9E9, 9E9, 9E9]];
    CONST robtarget p13111:= [[1505.6862847584605, 61.61126558902593, 1004.500033578516], [0, 0, 1, 0], [0, 0, 0, 0], [9E9, 9E9, 9E9, 9E9, 9E9, 9E9]];
    CONST robtarget p13112:= [[1506.2891513926352, 61.57437498457021, 1004.500033578516], [0, 0, 1, 0], [0, 0, 0, 0], [9E9, 9E9, 9E9, 9E9, 9E9, 9E9]];
    CONST robtarget p13113:= [[1506.663090986015, 61.566727134741356, 1004.500033578516], [0, 0, 1, 0], [0, 0, 0, 0], [9E9, 9E9, 9E9, 9E9, 9E9, 9E9]];
    CONST robtarget p13114:= [[1506.7295031757758, 61.55640393859453, 1004.500033578516], [0, 0, 1, 0], [0, 0, 0, 0], [9E9, 9E9, 9E9, 9E9, 9E9, 9E9]];
    CONST robtarget p13115:= [[1507.1395243097113, 61.49734047518008, 1004.500033578516], [0, 0, 1, 0], [0, 0, 0, 0], [9E9, 9E9, 9E9, 9E9, 9E9, 9E9]];
    CONST robtarget p13116:= [[1507.5619818505802, 61.44437926805831, 1004.500033578516], [0, 0, 1, 0], [0, 0, 0, 0], [9E9, 9E9, 9E9, 9E9, 9E9, 9E9]];
    CONST robtarget p13117:= [[1507.7930486831472, 61.40409988452909, 1004.500033578516], [0, 0, 1, 0], [0, 0, 0, 0], [9E9, 9E9, 9E9, 9E9, 9E9, 9E9]];
    CONST robtarget p13118:= [[1508.9656003014504, 61.23994250699515, 1004.500033578516], [0, 0, 1, 0], [0, 0, 0, 0], [9E9, 9E9, 9E9, 9E9, 9E9, 9E9]];
    CONST robtarget p13119:= [[1509.0824139648291, 61.21912038723799, 1004.500033578516], [0, 0, 1, 0], [0, 0, 0, 0], [9E9, 9E9, 9E9, 9E9, 9E9, 9E9]];
    CONST robtarget p13120:= [[1509.8416177771715, 61.095666097246394, 1004.500033578516], [0, 0, 1, 0], [0, 0, 0, 0], [9E9, 9E9, 9E9, 9E9, 9E9, 9E9]];
    CONST robtarget p13121:= [[1510.6698599607635, 60.94851958306951, 1004.500033578516], [0, 0, 1, 0], [0, 0, 0, 0], [9E9, 9E9, 9E9, 9E9, 9E9, 9E9]];
    CONST robtarget p13122:= [[1511.0853094035383, 60.887662595005466, 1004.500033578516], [0, 0, 1, 0], [0, 0, 0, 0], [9E9, 9E9, 9E9, 9E9, 9E9, 9E9]];
    CONST robtarget p13123:= [[1511.5280302307694, 60.84256056220839, 1004.500033578516], [0, 0, 1, 0], [0, 0, 0, 0], [9E9, 9E9, 9E9, 9E9, 9E9, 9E9]];
    CONST robtarget p13124:= [[1511.6156458802805, 60.8211553351192, 1004.500033578516], [0, 0, 1, 0], [0, 0, 0, 0], [9E9, 9E9, 9E9, 9E9, 9E9, 9E9]];
    CONST robtarget p13125:= [[1512.154768292444, 60.703590325900294, 1004.500033578516], [0, 0, 1, 0], [0, 0, 0, 0], [9E9, 9E9, 9E9, 9E9, 9E9, 9E9]];
    CONST robtarget p13126:= [[1513.0642657098952, 60.49770579297363, 1004.500033578516], [0, 0, 1, 0], [0, 0, 0, 0], [9E9, 9E9, 9E9, 9E9, 9E9, 9E9]];
    CONST robtarget p13127:= [[1513.6363952373422, 60.35311172546024, 1004.500033578516], [0, 0, 1, 0], [0, 0, 0, 0], [9E9, 9E9, 9E9, 9E9, 9E9, 9E9]];
    CONST robtarget p13128:= [[1514.0751095287965, 60.25725689202589, 1004.500033578516], [0, 0, 1, 0], [0, 0, 0, 0], [9E9, 9E9, 9E9, 9E9, 9E9, 9E9]];
    CONST robtarget p13129:= [[1514.349249033629, 60.21091255621319, 1004.500033578516], [0, 0, 1, 0], [0, 0, 0, 0], [9E9, 9E9, 9E9, 9E9, 9E9, 9E9]];
    CONST robtarget p13130:= [[1515.137220871783, 59.99669719651523, 1004.500033578516], [0, 0, 1, 0], [0, 0, 0, 0], [9E9, 9E9, 9E9, 9E9, 9E9, 9E9]];
    CONST robtarget p13131:= [[1515.6851765312454, 59.87418625272723, 1004.500033578516], [0, 0, 1, 0], [0, 0, 0, 0], [9E9, 9E9, 9E9, 9E9, 9E9, 9E9]];
    CONST robtarget p13132:= [[1516.0984783501224, 59.77904613678386, 1004.500033578516], [0, 0, 1, 0], [0, 0, 0, 0], [9E9, 9E9, 9E9, 9E9, 9E9, 9E9]];
    CONST robtarget p13133:= [[1516.4982182550077, 59.65795964116863, 1004.500033578516], [0, 0, 1, 0], [0, 0, 0, 0], [9E9, 9E9, 9E9, 9E9, 9E9, 9E9]];
    CONST robtarget p13134:= [[1517.1115315830964, 59.45600934598211, 1004.500033578516], [0, 0, 1, 0], [0, 0, 0, 0], [9E9, 9E9, 9E9, 9E9, 9E9, 9E9]];
    CONST robtarget p13135:= [[1517.4972523534657, 59.35586633975812, 1004.500033578516], [0, 0, 1, 0], [0, 0, 0, 0], [9E9, 9E9, 9E9, 9E9, 9E9, 9E9]];
    CONST robtarget p13136:= [[1518.1324390184595, 59.16512656520878, 1004.500033578516], [0, 0, 1, 0], [0, 0, 0, 0], [9E9, 9E9, 9E9, 9E9, 9E9, 9E9]];
    CONST robtarget p13137:= [[1518.3993225833672, 59.087324540796985, 1004.500033578516], [0, 0, 1, 0], [0, 0, 0, 0], [9E9, 9E9, 9E9, 9E9, 9E9, 9E9]];
    CONST robtarget p13138:= [[1519.4105585105312, 58.783146641539574, 1004.500033578516], [0, 0, 1, 0], [0, 0, 0, 0], [9E9, 9E9, 9E9, 9E9, 9E9, 9E9]];
    CONST robtarget p13139:= [[1519.8292393016918, 58.65935039396898, 1004.500033578516], [0, 0, 1, 0], [0, 0, 0, 0], [9E9, 9E9, 9E9, 9E9, 9E9, 9E9]];
    CONST robtarget p13140:= [[1520.211526363034, 58.52073181455664, 1004.500033578516], [0, 0, 1, 0], [0, 0, 0, 0], [9E9, 9E9, 9E9, 9E9, 9E9, 9E9]];
    CONST robtarget p13141:= [[1520.4987057546439, 58.4305717581277, 1004.500033578516], [0, 0, 1, 0], [0, 0, 0, 0], [9E9, 9E9, 9E9, 9E9, 9E9, 9E9]];
    CONST robtarget p13142:= [[1520.5745571116304, 58.40162081522858, 1004.500033578516], [0, 0, 1, 0], [0, 0, 0, 0], [9E9, 9E9, 9E9, 9E9, 9E9, 9E9]];
    CONST robtarget p13143:= [[1521.350029945068, 58.093994980819545, 1004.500033578516], [0, 0, 1, 0], [0, 0, 0, 0], [9E9, 9E9, 9E9, 9E9, 9E9, 9E9]];
    CONST robtarget p13144:= [[1521.8107612498939, 57.88460043539273, 1004.500033578516], [0, 0, 1, 0], [0, 0, 0, 0], [9E9, 9E9, 9E9, 9E9, 9E9, 9E9]];
    CONST robtarget p13145:= [[1522.304094750876, 57.713149571437256, 1004.500033578516], [0, 0, 1, 0], [0, 0, 0, 0], [9E9, 9E9, 9E9, 9E9, 9E9, 9E9]];
    CONST robtarget p13146:= [[1522.6450880823866, 57.58474411995843, 1004.500033578516], [0, 0, 1, 0], [0, 0, 0, 0], [9E9, 9E9, 9E9, 9E9, 9E9, 9E9]];
    CONST robtarget p13147:= [[1523.1495530033417, 57.40782845718205, 1004.500033578516], [0, 0, 1, 0], [0, 0, 0, 0], [9E9, 9E9, 9E9, 9E9, 9E9, 9E9]];
    CONST robtarget p13148:= [[1523.4438968577974, 57.30129190997184, 1004.500033578516], [0, 0, 1, 0], [0, 0, 0, 0], [9E9, 9E9, 9E9, 9E9, 9E9, 9E9]];
    CONST robtarget p13149:= [[1523.7951411061642, 57.155218725508135, 1004.500033578516], [0, 0, 1, 0], [0, 0, 0, 0], [9E9, 9E9, 9E9, 9E9, 9E9, 9E9]];
    CONST robtarget p13150:= [[1524.2100238897606, 56.958941661782404, 1004.500033578516], [0, 0, 1, 0], [0, 0, 0, 0], [9E9, 9E9, 9E9, 9E9, 9E9, 9E9]];
    CONST robtarget p13151:= [[1524.5186957242536, 56.839906257221315, 1004.500033578516], [0, 0, 1, 0], [0, 0, 0, 0], [9E9, 9E9, 9E9, 9E9, 9E9, 9E9]];
    CONST robtarget p13152:= [[1524.623220363781, 56.79620266390826, 1004.500033578516], [0, 0, 1, 0], [0, 0, 0, 0], [9E9, 9E9, 9E9, 9E9, 9E9, 9E9]];
    CONST robtarget p13153:= [[1524.9559505014277, 56.64055234732842, 1004.500033578516], [0, 0, 1, 0], [0, 0, 0, 0], [9E9, 9E9, 9E9, 9E9, 9E9, 9E9]];
    CONST robtarget p13154:= [[1525.1098299650937, 56.577083328930144, 1004.500033578516], [0, 0, 1, 0], [0, 0, 0, 0], [9E9, 9E9, 9E9, 9E9, 9E9, 9E9]];
    CONST robtarget p13155:= [[1525.3124227899705, 56.472019509201616, 1004.500033578516], [0, 0, 1, 0], [0, 0, 0, 0], [9E9, 9E9, 9E9, 9E9, 9E9, 9E9]];
    CONST robtarget p13156:= [[1525.637486329709, 56.323931445359364, 1004.500033578516], [0, 0, 1, 0], [0, 0, 0, 0], [9E9, 9E9, 9E9, 9E9, 9E9, 9E9]];
    CONST robtarget p13157:= [[1525.7743175754401, 56.2563037933122, 1004.500033578516], [0, 0, 1, 0], [0, 0, 0, 0], [9E9, 9E9, 9E9, 9E9, 9E9, 9E9]];
    CONST robtarget p13158:= [[1526.3476956271077, 56.00452333516316, 1004.500033578516], [0, 0, 1, 0], [0, 0, 0, 0], [9E9, 9E9, 9E9, 9E9, 9E9, 9E9]];
    CONST robtarget p13159:= [[1526.7424982778957, 55.80184233703662, 1004.500033578516], [0, 0, 1, 0], [0, 0, 0, 0], [9E9, 9E9, 9E9, 9E9, 9E9, 9E9]];
    CONST robtarget p13160:= [[1526.9418024051786, 55.71433551616202, 1004.500033578516], [0, 0, 1, 0], [0, 0, 0, 0], [9E9, 9E9, 9E9, 9E9, 9E9, 9E9]];
    CONST robtarget p13161:= [[1527.380240653982, 55.518617727321654, 1004.500033578516], [0, 0, 1, 0], [0, 0, 0, 0], [9E9, 9E9, 9E9, 9E9, 9E9, 9E9]];
    CONST robtarget p13162:= [[1527.7177509725784, 55.360843960503104, 1004.500033578516], [0, 0, 1, 0], [0, 0, 0, 0], [9E9, 9E9, 9E9, 9E9, 9E9, 9E9]];
    CONST robtarget p13163:= [[1528.1115118776966, 55.13316584402932, 1004.500033578516], [0, 0, 1, 0], [0, 0, 0, 0], [9E9, 9E9, 9E9, 9E9, 9E9, 9E9]];
    CONST robtarget p13164:= [[1528.656607150671, 54.8817568745434, 1004.500033578516], [0, 0, 1, 0], [0, 0, 0, 0], [9E9, 9E9, 9E9, 9E9, 9E9, 9E9]];
    CONST robtarget p13165:= [[1529.1916730770702, 54.571561269256904, 1004.500033578516], [0, 0, 1, 0], [0, 0, 0, 0], [9E9, 9E9, 9E9, 9E9, 9E9, 9E9]];
    CONST robtarget p13166:= [[1529.9344922608411, 54.16908478682785, 1004.500033578516], [0, 0, 1, 0], [0, 0, 0, 0], [9E9, 9E9, 9E9, 9E9, 9E9, 9E9]];
    CONST robtarget p13167:= [[1530.1136143911717, 54.069494438796326, 1004.500033578516], [0, 0, 1, 0], [0, 0, 0, 0], [9E9, 9E9, 9E9, 9E9, 9E9, 9E9]];
    CONST robtarget p13168:= [[1530.4934627343375, 53.864093596029704, 1004.500033578516], [0, 0, 1, 0], [0, 0, 0, 0], [9E9, 9E9, 9E9, 9E9, 9E9, 9E9]];
    CONST robtarget p13169:= [[1530.9678740843524, 53.55835012605681, 1004.500033578516], [0, 0, 1, 0], [0, 0, 0, 0], [9E9, 9E9, 9E9, 9E9, 9E9, 9E9]];
    CONST robtarget p13170:= [[1531.2807369583707, 53.39317443777496, 1004.500033578516], [0, 0, 1, 0], [0, 0, 0, 0], [9E9, 9E9, 9E9, 9E9, 9E9, 9E9]];
    CONST robtarget p13171:= [[1532.079312119388, 52.97160296012879, 1004.500033578516], [0, 0, 1, 0], [0, 0, 0, 0], [9E9, 9E9, 9E9, 9E9, 9E9, 9E9]];
    CONST robtarget p13172:= [[1532.1174435225744, 52.94758138972146, 1004.500033578516], [0, 0, 1, 0], [0, 0, 0, 0], [9E9, 9E9, 9E9, 9E9, 9E9, 9E9]];
    CONST robtarget p13173:= [[1532.4121324951602, 52.73595203111641, 1004.500033578516], [0, 0, 1, 0], [0, 0, 0, 0], [9E9, 9E9, 9E9, 9E9, 9E9, 9E9]];
    CONST robtarget p13174:= [[1532.7588593335386, 52.523757661538525, 1004.500033578516], [0, 0, 1, 0], [0, 0, 0, 0], [9E9, 9E9, 9E9, 9E9, 9E9, 9E9]];
    CONST robtarget p13175:= [[1533.2266480939556, 52.22212992442937, 1004.500033578516], [0, 0, 1, 0], [0, 0, 0, 0], [9E9, 9E9, 9E9, 9E9, 9E9, 9E9]];
    CONST robtarget p13176:= [[1533.8171335986854, 51.837510197977736, 1004.500033578516], [0, 0, 1, 0], [0, 0, 0, 0], [9E9, 9E9, 9E9, 9E9, 9E9, 9E9]];
    CONST robtarget p13177:= [[1533.9356095194703, 51.76513452300989, 1004.500033578516], [0, 0, 1, 0], [0, 0, 0, 0], [9E9, 9E9, 9E9, 9E9, 9E9, 9E9]];
    CONST robtarget p13178:= [[1534.968940098181, 51.03977915326402, 1004.500033578516], [0, 0, 1, 0], [0, 0, 0, 0], [9E9, 9E9, 9E9, 9E9, 9E9, 9E9]];
    CONST robtarget p13179:= [[1535.8063343513884, 50.51776578585675, 1004.500033578516], [0, 0, 1, 0], [0, 0, 0, 0], [9E9, 9E9, 9E9, 9E9, 9E9, 9E9]];
    CONST robtarget p13180:= [[1536.4707413175438, 49.9952312000716, 1004.500033578516], [0, 0, 1, 0], [0, 0, 0, 0], [9E9, 9E9, 9E9, 9E9, 9E9, 9E9]];
    CONST robtarget p13181:= [[1536.9162209570081, 49.68677118689742, 1004.500033578516], [0, 0, 1, 0], [0, 0, 0, 0], [9E9, 9E9, 9E9, 9E9, 9E9, 9E9]];
    CONST robtarget p13182:= [[1537.3466040362534, 49.34416467318404, 1004.500033578516], [0, 0, 1, 0], [0, 0, 0, 0], [9E9, 9E9, 9E9, 9E9, 9E9, 9E9]];
    CONST robtarget p13183:= [[1538.1160265790209, 48.75860319425175, 1004.500033578516], [0, 0, 1, 0], [0, 0, 0, 0], [9E9, 9E9, 9E9, 9E9, 9E9, 9E9]];
    CONST robtarget p13184:= [[1538.7788308217328, 48.241245716511074, 1004.500033578516], [0, 0, 1, 0], [0, 0, 0, 0], [9E9, 9E9, 9E9, 9E9, 9E9, 9E9]];
    CONST robtarget p13185:= [[1539.0399224290984, 48.04407934485009, 1004.500033578516], [0, 0, 1, 0], [0, 0, 0, 0], [9E9, 9E9, 9E9, 9E9, 9E9, 9E9]];
    CONST robtarget p13186:= [[1539.5677532968891, 47.64676920229533, 1004.500033578516], [0, 0, 1, 0], [0, 0, 0, 0], [9E9, 9E9, 9E9, 9E9, 9E9, 9E9]];
    CONST robtarget p13187:= [[1540.1447458205544, 47.1243555443601, 1004.500033578516], [0, 0, 1, 0], [0, 0, 0, 0], [9E9, 9E9, 9E9, 9E9, 9E9, 9E9]];
    CONST robtarget p13188:= [[1540.2781457856433, 47.00982049202486, 1004.500033578516], [0, 0, 1, 0], [0, 0, 0, 0], [9E9, 9E9, 9E9, 9E9, 9E9, 9E9]];
    CONST robtarget p13189:= [[1540.5481365264525, 46.76442821553087, 1004.500033578516], [0, 0, 1, 0], [0, 0, 0, 0], [9E9, 9E9, 9E9, 9E9, 9E9, 9E9]];
    CONST robtarget p13190:= [[1540.7921668783213, 46.523895946686196, 1004.500033578516], [0, 0, 1, 0], [0, 0, 0, 0], [9E9, 9E9, 9E9, 9E9, 9E9, 9E9]];
    CONST robtarget p13191:= [[1541.1206372424685, 46.234008623836075, 1004.500033578516], [0, 0, 1, 0], [0, 0, 0, 0], [9E9, 9E9, 9E9, 9E9, 9E9, 9E9]];
    CONST robtarget p13192:= [[1541.7623527793335, 45.685025726744286, 1004.500033578516], [0, 0, 1, 0], [0, 0, 0, 0], [9E9, 9E9, 9E9, 9E9, 9E9, 9E9]];
    CONST robtarget p13193:= [[1542.0958071655548, 45.3781630001111, 1004.500033578516], [0, 0, 1, 0], [0, 0, 0, 0], [9E9, 9E9, 9E9, 9E9, 9E9, 9E9]];
    CONST robtarget p13194:= [[1542.3250135127282, 45.171121329369, 1004.500033578516], [0, 0, 1, 0], [0, 0, 0, 0], [9E9, 9E9, 9E9, 9E9, 9E9, 9E9]];
    CONST robtarget p13195:= [[1542.5426172092716, 44.96456027617546, 1004.500033578516], [0, 0, 1, 0], [0, 0, 0, 0], [9E9, 9E9, 9E9, 9E9, 9E9, 9E9]];
    CONST robtarget p13196:= [[1543.1020468462627, 44.442593094868215, 1004.500033578516], [0, 0, 1, 0], [0, 0, 0, 0], [9E9, 9E9, 9E9, 9E9, 9E9, 9E9]];
    CONST robtarget p13197:= [[1543.4261624588194, 44.10298138110426, 1004.500033578516], [0, 0, 1, 0], [0, 0, 0, 0], [9E9, 9E9, 9E9, 9E9, 9E9, 9E9]];
    CONST robtarget p13198:= [[1543.897329539247, 43.62426558363555, 1004.500033578516], [0, 0, 1, 0], [0, 0, 0, 0], [9E9, 9E9, 9E9, 9E9, 9E9, 9E9]];
    CONST robtarget p13199:= [[1544.1891416870783, 43.3219955539563, 1004.500033578516], [0, 0, 1, 0], [0, 0, 0, 0], [9E9, 9E9, 9E9, 9E9, 9E9, 9E9]];
    CONST robtarget p13200:= [[1544.5460645492, 42.93991877533189, 1004.500033578516], [0, 0, 1, 0], [0, 0, 0, 0], [9E9, 9E9, 9E9, 9E9, 9E9, 9E9]];
    CONST robtarget p13201:= [[1544.8336146163215, 42.647991439248926, 1004.500033578516], [0, 0, 1, 0], [0, 0, 0, 0], [9E9, 9E9, 9E9, 9E9, 9E9, 9E9]];
    CONST robtarget p13202:= [[1545.1006890920462, 42.35299912675376, 1004.500033578516], [0, 0, 1, 0], [0, 0, 0, 0], [9E9, 9E9, 9E9, 9E9, 9E9, 9E9]];
    CONST robtarget p13203:= [[1545.5396921324138, 41.850406730972836, 1004.500033578516], [0, 0, 1, 0], [0, 0, 0, 0], [9E9, 9E9, 9E9, 9E9, 9E9, 9E9]];
    CONST robtarget p13204:= [[1545.6436742209194, 41.73918811182179, 1004.500033578516], [0, 0, 1, 0], [0, 0, 0, 0], [9E9, 9E9, 9E9, 9E9, 9E9, 9E9]];
    CONST robtarget p13205:= [[1546.2271876212374, 41.19968837856081, 1004.500033578516], [0, 0, 1, 0], [0, 0, 0, 0], [9E9, 9E9, 9E9, 9E9, 9E9, 9E9]];
    CONST robtarget p13206:= [[1546.4425754311496, 40.950150844029736, 1004.500033578516], [0, 0, 1, 0], [0, 0, 0, 0], [9E9, 9E9, 9E9, 9E9, 9E9, 9E9]];
    CONST robtarget p13207:= [[1547.0866818213817, 40.18074002118168, 1004.500033578516], [0, 0, 1, 0], [0, 0, 0, 0], [9E9, 9E9, 9E9, 9E9, 9E9, 9E9]];
    CONST robtarget p13208:= [[1547.4990168583727, 39.65510971783576, 1004.500033578516], [0, 0, 1, 0], [0, 0, 0, 0], [9E9, 9E9, 9E9, 9E9, 9E9, 9E9]];
    CONST robtarget p13209:= [[1547.6307487659205, 39.51323963427356, 1004.500033578516], [0, 0, 1, 0], [0, 0, 0, 0], [9E9, 9E9, 9E9, 9E9, 9E9, 9E9]];
    CONST robtarget p13210:= [[1547.8271765553768, 39.282546689421196, 1004.500033578516], [0, 0, 1, 0], [0, 0, 0, 0], [9E9, 9E9, 9E9, 9E9, 9E9, 9E9]];
    CONST robtarget p13211:= [[1548.2292099843964, 38.78116576695639, 1004.500033578516], [0, 0, 1, 0], [0, 0, 0, 0], [9E9, 9E9, 9E9, 9E9, 9E9, 9E9]];
    CONST robtarget p13212:= [[1548.5775737178762, 38.38499435456002, 1004.500033578516], [0, 0, 1, 0], [0, 0, 0, 0], [9E9, 9E9, 9E9, 9E9, 9E9, 9E9]];
    CONST robtarget p13213:= [[1548.9315504193983, 37.82503695771294, 1004.500033578516], [0, 0, 1, 0], [0, 0, 0, 0], [9E9, 9E9, 9E9, 9E9, 9E9, 9E9]];
    CONST robtarget p13214:= [[1549.2101318954922, 37.47655557532454, 1004.500033578516], [0, 0, 1, 0], [0, 0, 0, 0], [9E9, 9E9, 9E9, 9E9, 9E9, 9E9]];
    CONST robtarget p13215:= [[1549.3652428327057, 37.297010054613736, 1004.500033578516], [0, 0, 1, 0], [0, 0, 0, 0], [9E9, 9E9, 9E9, 9E9, 9E9, 9E9]];
    CONST robtarget p13216:= [[1549.5605179908853, 37.02215705142362, 1004.500033578516], [0, 0, 1, 0], [0, 0, 0, 0], [9E9, 9E9, 9E9, 9E9, 9E9, 9E9]];
    CONST robtarget p13217:= [[1550.225385683209, 36.13025157464817, 1004.500033578516], [0, 0, 1, 0], [0, 0, 0, 0], [9E9, 9E9, 9E9, 9E9, 9E9, 9E9]];
    CONST robtarget p13218:= [[1550.5360993979093, 35.6946754328922, 1004.500033578516], [0, 0, 1, 0], [0, 0, 0, 0], [9E9, 9E9, 9E9, 9E9, 9E9, 9E9]];
    CONST robtarget p13219:= [[1550.8767348423642, 35.22356066994553, 1004.500033578516], [0, 0, 1, 0], [0, 0, 0, 0], [9E9, 9E9, 9E9, 9E9, 9E9, 9E9]];
    CONST robtarget p13220:= [[1551.2299297693007, 34.73723243984132, 1004.500033578516], [0, 0, 1, 0], [0, 0, 0, 0], [9E9, 9E9, 9E9, 9E9, 9E9, 9E9]];
    CONST robtarget p13221:= [[1551.5528398551871, 34.30616304150534, 1004.500033578516], [0, 0, 1, 0], [0, 0, 0, 0], [9E9, 9E9, 9E9, 9E9, 9E9, 9E9]];
    CONST robtarget p13222:= [[1551.5595596693986, 34.29323463321808, 1004.500033578516], [0, 0, 1, 0], [0, 0, 0, 0], [9E9, 9E9, 9E9, 9E9, 9E9, 9E9]];
    CONST robtarget p13223:= [[1551.8584744233538, 33.76869450067305, 1004.500033578516], [0, 0, 1, 0], [0, 0, 0, 0], [9E9, 9E9, 9E9, 9E9, 9E9, 9E9]];
    CONST robtarget p13224:= [[1552.2000278163243, 33.24327855605077, 1004.500033578516], [0, 0, 1, 0], [0, 0, 0, 0], [9E9, 9E9, 9E9, 9E9, 9E9, 9E9]];
    CONST robtarget p13225:= [[1552.3165469372975, 33.05423581701322, 1004.500033578516], [0, 0, 1, 0], [0, 0, 0, 0], [9E9, 9E9, 9E9, 9E9, 9E9, 9E9]];
    CONST robtarget p13226:= [[1552.4962637578271, 32.78867543261707, 1004.500033578516], [0, 0, 1, 0], [0, 0, 0, 0], [9E9, 9E9, 9E9, 9E9, 9E9, 9E9]];
    CONST robtarget p13227:= [[1552.9272742581693, 32.08450881490957, 1004.500033578516], [0, 0, 1, 0], [0, 0, 0, 0], [9E9, 9E9, 9E9, 9E9, 9E9, 9E9]];
    CONST robtarget p13228:= [[1553.1427924987202, 31.700756333050663, 1004.500033578516], [0, 0, 1, 0], [0, 0, 0, 0], [9E9, 9E9, 9E9, 9E9, 9E9, 9E9]];
    CONST robtarget p13229:= [[1553.3212197811708, 31.406304580094414, 1004.500033578516], [0, 0, 1, 0], [0, 0, 0, 0], [9E9, 9E9, 9E9, 9E9, 9E9, 9E9]];
    CONST robtarget p13230:= [[1553.6434838514442, 30.884741035014528, 1004.500033578516], [0, 0, 1, 0], [0, 0, 0, 0], [9E9, 9E9, 9E9, 9E9, 9E9, 9E9]];
    CONST robtarget p13231:= [[1553.804278913582, 30.618928213454765, 1004.500033578516], [0, 0, 1, 0], [0, 0, 0, 0], [9E9, 9E9, 9E9, 9E9, 9E9, 9E9]];
    CONST robtarget p13232:= [[1554.002378814152, 30.319424070646676, 1004.500033578516], [0, 0, 1, 0], [0, 0, 0, 0], [9E9, 9E9, 9E9, 9E9, 9E9, 9E9]];
    CONST robtarget p13233:= [[1554.4488142142593, 29.37112240387775, 1004.500033578516], [0, 0, 1, 0], [0, 0, 0, 0], [9E9, 9E9, 9E9, 9E9, 9E9, 9E9]];
    CONST robtarget p13234:= [[1554.8045574052433, 28.754681749196507, 1004.500033578516], [0, 0, 1, 0], [0, 0, 0, 0], [9E9, 9E9, 9E9, 9E9, 9E9, 9E9]];
    CONST robtarget p13235:= [[1555.1810781360687, 27.948583690423916, 1004.500033578516], [0, 0, 1, 0], [0, 0, 0, 0], [9E9, 9E9, 9E9, 9E9, 9E9, 9E9]];
    CONST robtarget p13236:= [[1555.433432285193, 27.499525543202054, 1004.500033578516], [0, 0, 1, 0], [0, 0, 0, 0], [9E9, 9E9, 9E9, 9E9, 9E9, 9E9]];
    CONST robtarget p13237:= [[1555.515257304809, 27.34712472939819, 1004.500033578516], [0, 0, 1, 0], [0, 0, 0, 0], [9E9, 9E9, 9E9, 9E9, 9E9, 9E9]];
    CONST robtarget p13238:= [[1555.725319564946, 26.960815010380216, 1004.500033578516], [0, 0, 1, 0], [0, 0, 0, 0], [9E9, 9E9, 9E9, 9E9, 9E9, 9E9]];
    CONST robtarget p13239:= [[1555.8477072878861, 26.730490763758638, 1004.500033578516], [0, 0, 1, 0], [0, 0, 0, 0], [9E9, 9E9, 9E9, 9E9, 9E9, 9E9]];
    CONST robtarget p13240:= [[1556.0804484721461, 26.208439012312297, 1004.500033578516], [0, 0, 1, 0], [0, 0, 0, 0], [9E9, 9E9, 9E9, 9E9, 9E9, 9E9]];
    CONST robtarget p13241:= [[1556.2908442209773, 25.717092689298113, 1004.500033578516], [0, 0, 1, 0], [0, 0, 0, 0], [9E9, 9E9, 9E9, 9E9, 9E9, 9E9]];
    CONST robtarget p13242:= [[1556.4564360749755, 25.347869261736392, 1004.500033578516], [0, 0, 1, 0], [0, 0, 0, 0], [9E9, 9E9, 9E9, 9E9, 9E9, 9E9]];
    CONST robtarget p13243:= [[1556.633500575827, 24.957572774064246, 1004.500033578516], [0, 0, 1, 0], [0, 0, 0, 0], [9E9, 9E9, 9E9, 9E9, 9E9, 9E9]];
    CONST robtarget p13244:= [[1556.8017730997008, 24.55315329949613, 1004.500033578516], [0, 0, 1, 0], [0, 0, 0, 0], [9E9, 9E9, 9E9, 9E9, 9E9, 9E9]];
    CONST robtarget p13245:= [[1556.884275746069, 24.328510077042452, 1004.500033578516], [0, 0, 1, 0], [0, 0, 0, 0], [9E9, 9E9, 9E9, 9E9, 9E9, 9E9]];
    CONST robtarget p13246:= [[1557.2096914428619, 23.56482626543165, 1004.500033578516], [0, 0, 1, 0], [0, 0, 0, 0], [9E9, 9E9, 9E9, 9E9, 9E9, 9E9]];
    CONST robtarget p13247:= [[1557.4903566461383, 22.878760455235494, 1004.500033578516], [0, 0, 1, 0], [0, 0, 0, 0], [9E9, 9E9, 9E9, 9E9, 9E9, 9E9]];
    CONST robtarget p13248:= [[1557.8268737705073, 22.161100061330302, 1004.500033578516], [0, 0, 1, 0], [0, 0, 0, 0], [9E9, 9E9, 9E9, 9E9, 9E9, 9E9]];
    CONST robtarget p13249:= [[1557.8935069690067, 21.917885002054987, 1004.500033578516], [0, 0, 1, 0], [0, 0, 0, 0], [9E9, 9E9, 9E9, 9E9, 9E9, 9E9]];
    CONST robtarget p13250:= [[1558.2103807776662, 21.03451382422709, 1004.500033578516], [0, 0, 1, 0], [0, 0, 0, 0], [9E9, 9E9, 9E9, 9E9, 9E9, 9E9]];
    CONST robtarget p13251:= [[1558.4705760538307, 20.243022849098224, 1004.500033578516], [0, 0, 1, 0], [0, 0, 0, 0], [9E9, 9E9, 9E9, 9E9, 9E9, 9E9]];
    CONST robtarget p13252:= [[1558.5293826005086, 20.097698604475127, 1004.500033578516], [0, 0, 1, 0], [0, 0, 0, 0], [9E9, 9E9, 9E9, 9E9, 9E9, 9E9]];
    CONST robtarget p13253:= [[1558.7448614921761, 19.417284089288472, 1004.500033578516], [0, 0, 1, 0], [0, 0, 0, 0], [9E9, 9E9, 9E9, 9E9, 9E9, 9E9]];
    CONST robtarget p13254:= [[1558.9811728967638, 18.725781480095804, 1004.500033578516], [0, 0, 1, 0], [0, 0, 0, 0], [9E9, 9E9, 9E9, 9E9, 9E9, 9E9]];
    CONST robtarget p13255:= [[1559.1485636435118, 18.291065578263698, 1004.500033578516], [0, 0, 1, 0], [0, 0, 0, 0], [9E9, 9E9, 9E9, 9E9, 9E9, 9E9]];
    CONST robtarget p13256:= [[1559.2440371857645, 18.01995734792517, 1004.500033578516], [0, 0, 1, 0], [0, 0, 0, 0], [9E9, 9E9, 9E9, 9E9, 9E9, 9E9]];
    CONST robtarget p13257:= [[1559.379251402489, 17.542110190374018, 1004.500033578516], [0, 0, 1, 0], [0, 0, 0, 0], [9E9, 9E9, 9E9, 9E9, 9E9, 9E9]];
    CONST robtarget p13258:= [[1559.5039739294068, 17.095945380772136, 1004.500033578516], [0, 0, 1, 0], [0, 0, 0, 0], [9E9, 9E9, 9E9, 9E9, 9E9, 9E9]];
    CONST robtarget p13259:= [[1559.7570263642972, 16.128476733276514, 1004.500033578516], [0, 0, 1, 0], [0, 0, 0, 0], [9E9, 9E9, 9E9, 9E9, 9E9, 9E9]];
    CONST robtarget p13260:= [[1559.8050151818375, 15.879465453284539, 1004.500033578516], [0, 0, 1, 0], [0, 0, 0, 0], [9E9, 9E9, 9E9, 9E9, 9E9, 9E9]];
    CONST robtarget p13261:= [[1560.020475538835, 15.081426431490982, 1004.500033578516], [0, 0, 1, 0], [0, 0, 0, 0], [9E9, 9E9, 9E9, 9E9, 9E9, 9E9]];
    CONST robtarget p13262:= [[1560.180473771669, 14.365764823758497, 1004.500033578516], [0, 0, 1, 0], [0, 0, 0, 0], [9E9, 9E9, 9E9, 9E9, 9E9, 9E9]];
    CONST robtarget p13263:= [[1560.3832289108511, 13.737331305648851, 1004.500033578516], [0, 0, 1, 0], [0, 0, 0, 0], [9E9, 9E9, 9E9, 9E9, 9E9, 9E9]];
    CONST robtarget p13264:= [[1560.5406918719052, 12.974564534769783, 1004.500033578516], [0, 0, 1, 0], [0, 0, 0, 0], [9E9, 9E9, 9E9, 9E9, 9E9, 9E9]];
    CONST robtarget p13265:= [[1560.639631157924, 12.417614318478101, 1004.500033578516], [0, 0, 1, 0], [0, 0, 0, 0], [9E9, 9E9, 9E9, 9E9, 9E9, 9E9]];
    CONST robtarget p13266:= [[1560.6681834540714, 12.240206118687198, 1004.500033578516], [0, 0, 1, 0], [0, 0, 0, 0], [9E9, 9E9, 9E9, 9E9, 9E9, 9E9]];
    CONST robtarget p13267:= [[1560.8129704764892, 11.450536931470353, 1004.500033578516], [0, 0, 1, 0], [0, 0, 0, 0], [9E9, 9E9, 9E9, 9E9, 9E9, 9E9]];
    CONST robtarget p13268:= [[1560.9538391733201, 10.758162921692673, 1004.500033578516], [0, 0, 1, 0], [0, 0, 0, 0], [9E9, 9E9, 9E9, 9E9, 9E9, 9E9]];
    CONST robtarget p13269:= [[1560.964941648623, 10.671417326389914, 1004.500033578516], [0, 0, 1, 0], [0, 0, 0, 0], [9E9, 9E9, 9E9, 9E9, 9E9, 9E9]];
    CONST robtarget p13270:= [[1561.0007483341967, 10.365976332514904, 1004.500033578516], [0, 0, 1, 0], [0, 0, 0, 0], [9E9, 9E9, 9E9, 9E9, 9E9, 9E9]];
    CONST robtarget p13271:= [[1561.1659645083369, 9.448178493671705, 1004.500033578516], [0, 0, 1, 0], [0, 0, 0, 0], [9E9, 9E9, 9E9, 9E9, 9E9, 9E9]];
    CONST robtarget p13272:= [[1561.192517816966, 9.313063348400846, 1004.500033578516], [0, 0, 1, 0], [0, 0, 0, 0], [9E9, 9E9, 9E9, 9E9, 9E9, 9E9]];
    CONST robtarget p13273:= [[1561.2399908188781, 9.08353192111204, 1004.500033578516], [0, 0, 1, 0], [0, 0, 0, 0], [9E9, 9E9, 9E9, 9E9, 9E9, 9E9]];
    CONST robtarget p13274:= [[1561.2876219034265, 8.894336944504204, 1004.500033578516], [0, 0, 1, 0], [0, 0, 0, 0], [9E9, 9E9, 9E9, 9E9, 9E9, 9E9]];
    CONST robtarget p13275:= [[1561.3660389591396, 7.911961662908851, 1004.500033578516], [0, 0, 1, 0], [0, 0, 0, 0], [9E9, 9E9, 9E9, 9E9, 9E9, 9E9]];
    CONST robtarget p13276:= [[1561.4049665039745, 7.537642821677267, 1004.500033578516], [0, 0, 1, 0], [0, 0, 0, 0], [9E9, 9E9, 9E9, 9E9, 9E9, 9E9]];
    CONST robtarget p13277:= [[1561.4466760919606, 7.190691256846463, 1004.500033578516], [0, 0, 1, 0], [0, 0, 0, 0], [9E9, 9E9, 9E9, 9E9, 9E9, 9E9]];
    CONST robtarget p13278:= [[1561.5466217975704, 6.4988337487471455, 1004.500033578516], [0, 0, 1, 0], [0, 0, 0, 0], [9E9, 9E9, 9E9, 9E9, 9E9, 9E9]];
    CONST robtarget p13279:= [[1561.616633359475, 5.8158573486341965, 1004.500033578516], [0, 0, 1, 0], [0, 0, 0, 0], [9E9, 9E9, 9E9, 9E9, 9E9, 9E9]];
    CONST robtarget p13280:= [[1561.6792896576112, 5.213928844041476, 1004.500033578516], [0, 0, 1, 0], [0, 0, 0, 0], [9E9, 9E9, 9E9, 9E9, 9E9, 9E9]];
    CONST robtarget p13281:= [[1561.7250746607785, 4.773703215850034, 1004.500033578516], [0, 0, 1, 0], [0, 0, 0, 0], [9E9, 9E9, 9E9, 9E9, 9E9, 9E9]];
    CONST robtarget p13282:= [[1561.7523104153015, 4.257488955576079, 1004.500033578516], [0, 0, 1, 0], [0, 0, 0, 0], [9E9, 9E9, 9E9, 9E9, 9E9, 9E9]];
    CONST robtarget p13283:= [[1561.7638141167708, 4.084033824531247, 1004.500033578516], [0, 0, 1, 0], [0, 0, 0, 0], [9E9, 9E9, 9E9, 9E9, 9E9, 9E9]];
    CONST robtarget p13284:= [[1561.7973075556602, 3.6080452509004743, 1004.500033578516], [0, 0, 1, 0], [0, 0, 0, 0], [9E9, 9E9, 9E9, 9E9, 9E9, 9E9]];
    CONST robtarget p13285:= [[1561.8067797723606, 3.3097070648990012, 1004.500033578516], [0, 0, 1, 0], [0, 0, 0, 0], [9E9, 9E9, 9E9, 9E9, 9E9, 9E9]];
    CONST robtarget p13286:= [[1561.822158680893, 2.9098616991937263, 1004.500033578516], [0, 0, 1, 0], [0, 0, 0, 0], [9E9, 9E9, 9E9, 9E9, 9E9, 9E9]];
    CONST robtarget p13287:= [[1561.825353713137, 2.420323887888017, 1004.500033578516], [0, 0, 1, 0], [0, 0, 0, 0], [9E9, 9E9, 9E9, 9E9, 9E9, 9E9]];
    CONST robtarget p13288:= [[1561.8563014956333, 1.421575358975673, 1004.500033578516], [0, 0, 1, 0], [0, 0, 0, 0], [9E9, 9E9, 9E9, 9E9, 9E9, 9E9]];
    CONST robtarget p13289:= [[1561.8907158616496, 0.5495357864304538, 1004.500033578516], [0, 0, 1, 0], [0, 0, 0, 0], [9E9, 9E9, 9E9, 9E9, 9E9, 9E9]];
    CONST robtarget p13290:= [[1561.8988141801558, 0.47016391785209066, 1004.500033578516], [0, 0, 1, 0], [0, 0, 0, 0], [9E9, 9E9, 9E9, 9E9, 9E9, 9E9]];
    CONST robtarget p13291:= [[1561.8950477205249, 0.27055351615759093, 1004.500033578516], [0, 0, 1, 0], [0, 0, 0, 0], [9E9, 9E9, 9E9, 9E9, 9E9, 9E9]];
    CONST robtarget p13292:= [[1561.8926058631594, -0.052035899161168686, 1004.500033578516], [0, 0, 1, 0], [0, 0, 0, 0], [9E9, 9E9, 9E9, 9E9, 9E9, 9E9]];
    CONST robtarget p13293:= [[1561.8848896615118, -1.2492412908985813, 1004.500033578516], [0, 0, 1, 0], [0, 0, 0, 0], [9E9, 9E9, 9E9, 9E9, 9E9, 9E9]];
    CONST robtarget p13294:= [[1561.850031867312, -2.102968017445093, 1004.500033578516], [0, 0, 1, 0], [0, 0, 0, 0], [9E9, 9E9, 9E9, 9E9, 9E9, 9E9]];
    CONST robtarget p13295:= [[1561.8184583917136, -3.017242933688493, 1004.500033578516], [0, 0, 1, 0], [0, 0, 0, 0], [9E9, 9E9, 9E9, 9E9, 9E9, 9E9]];
    CONST robtarget p13296:= [[1561.8130978656645, -3.0589342500684467, 1004.500033578516], [0, 0, 1, 0], [0, 0, 0, 0], [9E9, 9E9, 9E9, 9E9, 9E9, 9E9]];
    CONST robtarget p13297:= [[1561.7665940346758, -3.6733798977280827, 1004.500033578516], [0, 0, 1, 0], [0, 0, 0, 0], [9E9, 9E9, 9E9, 9E9, 9E9, 9E9]];
    CONST robtarget p13298:= [[1561.727480535751, -4.434642757637235, 1004.500033578516], [0, 0, 1, 0], [0, 0, 0, 0], [9E9, 9E9, 9E9, 9E9, 9E9, 9E9]];
    CONST robtarget p13299:= [[1561.7325834757914, -4.666758570162344, 1004.500033578516], [0, 0, 1, 0], [0, 0, 0, 0], [9E9, 9E9, 9E9, 9E9, 9E9, 9E9]];
    CONST robtarget p13300:= [[1561.6361501929414, -5.221595033413337, 1004.500033578516], [0, 0, 1, 0], [0, 0, 0, 0], [9E9, 9E9, 9E9, 9E9, 9E9, 9E9]];
    CONST robtarget p13301:= [[1561.6235633143747, -5.322421621923098, 1004.500033578516], [0, 0, 1, 0], [0, 0, 0, 0], [9E9, 9E9, 9E9, 9E9, 9E9, 9E9]];
    CONST robtarget p13302:= [[1561.5584777032245, -6.119559254691623, 1004.500033578516], [0, 0, 1, 0], [0, 0, 0, 0], [9E9, 9E9, 9E9, 9E9, 9E9, 9E9]];
    CONST robtarget p13303:= [[1561.5560296044132, -6.320659656616051, 1004.500033578516], [0, 0, 1, 0], [0, 0, 0, 0], [9E9, 9E9, 9E9, 9E9, 9E9, 9E9]];
    CONST robtarget p13304:= [[1561.5349676904443, -6.521238988825523, 1004.500033578516], [0, 0, 1, 0], [0, 0, 0, 0], [9E9, 9E9, 9E9, 9E9, 9E9, 9E9]];
    CONST robtarget p13305:= [[1561.4806189585918, -6.9429147656584576, 1004.500033578516], [0, 0, 1, 0], [0, 0, 0, 0], [9E9, 9E9, 9E9, 9E9, 9E9, 9E9]];
    CONST robtarget p13306:= [[1561.422257088692, -7.505858223972091, 1004.500033578516], [0, 0, 1, 0], [0, 0, 0, 0], [9E9, 9E9, 9E9, 9E9, 9E9, 9E9]];
    CONST robtarget p13307:= [[1561.4109003353665, -7.760128204293366, 1004.500033578516], [0, 0, 1, 0], [0, 0, 0, 0], [9E9, 9E9, 9E9, 9E9, 9E9, 9E9]];
    CONST robtarget p13308:= [[1561.324122891428, -8.405568241628345, 1004.500033578516], [0, 0, 1, 0], [0, 0, 0, 0], [9E9, 9E9, 9E9, 9E9, 9E9, 9E9]];
    CONST robtarget p13309:= [[1561.2750802373869, -8.810427911946526, 1004.500033578516], [0, 0, 1, 0], [0, 0, 0, 0], [9E9, 9E9, 9E9, 9E9, 9E9, 9E9]];
    CONST robtarget p13310:= [[1561.1828318670218, -9.440872611760192, 1004.500033578516], [0, 0, 1, 0], [0, 0, 0, 0], [9E9, 9E9, 9E9, 9E9, 9E9, 9E9]];
    CONST robtarget p13311:= [[1561.161893635805, -9.608825018124563, 1004.500033578516], [0, 0, 1, 0], [0, 0, 0, 0], [9E9, 9E9, 9E9, 9E9, 9E9, 9E9]];
    CONST robtarget p13312:= [[1561.072773664851, -9.89902472208881, 1004.500033578516], [0, 0, 1, 0], [0, 0, 0, 0], [9E9, 9E9, 9E9, 9E9, 9E9, 9E9]];
    CONST robtarget p13313:= [[1560.8863277978942, -10.91501034046145, 1004.500033578516], [0, 0, 1, 0], [0, 0, 0, 0], [9E9, 9E9, 9E9, 9E9, 9E9, 9E9]];
    CONST robtarget p13314:= [[1560.8686071801503, -11.210151605342944, 1004.500033578516], [0, 0, 1, 0], [0, 0, 0, 0], [9E9, 9E9, 9E9, 9E9, 9E9, 9E9]];
    CONST robtarget p13315:= [[1560.8415779321354, -11.356649672005332, 1004.500033578516], [0, 0, 1, 0], [0, 0, 0, 0], [9E9, 9E9, 9E9, 9E9, 9E9, 9E9]];
    CONST robtarget p13316:= [[1560.7325385860745, -11.9173079080741, 1004.500033578516], [0, 0, 1, 0], [0, 0, 0, 0], [9E9, 9E9, 9E9, 9E9, 9E9, 9E9]];
    CONST robtarget p13317:= [[1560.6435723420946, -12.326242023091531, 1004.500033578516], [0, 0, 1, 0], [0, 0, 0, 0], [9E9, 9E9, 9E9, 9E9, 9E9, 9E9]];
    CONST robtarget p13318:= [[1560.5435051538998, -12.97516897849092, 1004.500033578516], [0, 0, 1, 0], [0, 0, 0, 0], [9E9, 9E9, 9E9, 9E9, 9E9, 9E9]];
    CONST robtarget p13319:= [[1560.3674074456526, -13.700998781672062, 1004.500033578516], [0, 0, 1, 0], [0, 0, 0, 0], [9E9, 9E9, 9E9, 9E9, 9E9, 9E9]];
    CONST robtarget p13320:= [[1560.2450551250358, -14.267574457520944, 1004.500033578516], [0, 0, 1, 0], [0, 0, 0, 0], [9E9, 9E9, 9E9, 9E9, 9E9, 9E9]];
    CONST robtarget p13321:= [[1559.9232578073445, -15.27833088725913, 1004.500033578516], [0, 0, 1, 0], [0, 0, 0, 0], [9E9, 9E9, 9E9, 9E9, 9E9, 9E9]];
    CONST robtarget p13322:= [[1559.821394727859, -15.737234241708208, 1004.500033578516], [0, 0, 1, 0], [0, 0, 0, 0], [9E9, 9E9, 9E9, 9E9, 9E9, 9E9]];
